C03563=1013.898,264.912,-139.732,168.814,53.259,160.172
C03564=1013.893,264.664,-139.704,168.809,53.267,160.173
C03565=1013.887,264.419,-139.676,168.803,53.274,160.173
C03566=1013.882,264.174,-139.648,168.798,53.282,160.174
C03567=1013.877,263.928,-139.620,168.793,53.290,160.175
C03568=1013.871,263.683,-139.592,168.787,53.298,160.175
C03569=1013.865,263.438,-139.565,168.782,53.306,160.176
C03570=1013.860,263.193,-139.538,168.777,53.313,160.177
C03571=1013.855,262.948,-139.510,168.772,53.321,160.177
C03572=1013.850,262.702,-139.482,168.766,53.329,160.178
C03573=1013.844,262.454,-139.454,168.762,53.337,160.179
C03574=1013.838,262.206,-139.426,168.756,53.346,160.179
C03575=1013.833,261.958,-139.398,168.751,53.353,160.180
C03576=1013.828,261.709,-139.371,168.746,53.361,160.181
C03577=1013.823,261.461,-139.343,168.740,53.369,160.181
C03578=1013.817,261.212,-139.315,168.735,53.377,160.182
C03579=1013.811,260.964,-139.287,168.729,53.386,160.183
C03580=1013.806,260.715,-139.259,168.725,53.393,160.183
C03581=1013.801,260.466,-139.231,168.719,53.402,160.184
C03582=1013.795,260.217,-139.203,168.714,53.410,160.185
C03583=1013.790,259.968,-139.175,168.708,53.418,160.185
C03584=1013.785,259.718,-139.147,168.703,53.426,160.186
C03585=1013.780,259.470,-139.119,168.699,53.434,160.187
C03586=1013.774,259.221,-139.092,168.693,53.443,160.188
C03587=1013.768,258.973,-139.064,168.687,53.451,160.188
C03588=1013.763,258.725,-139.037,168.682,53.459,160.189
C03589=1013.758,258.476,-139.011,168.677,53.468,160.190
C03590=1013.752,258.228,-138.983,168.672,53.476,160.191
C03591=1013.746,257.979,-138.956,168.666,53.484,160.191
C03592=1013.741,257.731,-138.928,168.662,53.492,160.192
C03593=1013.736,257.482,-138.900,168.656,53.501,160.193
C03594=1013.730,257.234,-138.874,168.651,53.509,160.194
C03595=1013.724,256.986,-138.846,168.646,53.518,160.194
C03596=1013.719,256.738,-138.819,168.640,53.526,160.195
C03597=1013.714,256.489,-138.792,168.635,53.534,160.196
C03598=1013.708,256.240,-138.764,168.630,53.543,160.197
C03599=1013.702,255.992,-138.737,168.625,53.551,160.197
C03600=1013.697,255.743,-138.710,168.620,53.560,160.198
C03601=1013.691,255.495,-138.683,168.614,53.568,160.199
C03602=1013.686,255.246,-138.656,168.610,53.576,160.200
C03603=1013.681,254.998,-138.629,168.604,53.585,160.200
C03604=1013.675,254.750,-138.601,168.599,53.593,160.201
C03605=1013.670,254.501,-138.574,168.594,53.602,160.202
C03606=1013.664,254.253,-138.547,168.589,53.610,160.203
C03607=1013.659,254.004,-138.520,168.583,53.619,160.204
C03608=1013.654,253.755,-138.493,168.578,53.628,160.204
C03609=1013.648,253.507,-138.466,168.573,53.635,160.205
C03610=1013.643,253.259,-138.438,168.568,53.644,160.206
C03611=1013.637,253.011,-138.412,168.562,53.653,160.207
C03612=1013.632,252.762,-138.384,168.558,53.661,160.208
C03613=1013.626,252.514,-138.358,168.552,53.670,160.208
C03614=1013.621,252.265,-138.330,168.548,53.678,160.209
C03615=1013.616,252.016,-138.303,168.542,53.687,160.210
C03616=1013.611,251.768,-138.276,168.537,53.696,160.211
C03617=1013.605,251.519,-138.249,168.532,53.704,160.212
C03618=1013.600,251.271,-138.223,168.527,53.713,160.212
C03619=1013.595,251.022,-138.195,168.522,53.721,160.213
C03620=1013.590,250.774,-138.168,168.517,53.730,160.214
C03621=1013.584,250.525,-138.141,168.511,53.739,160.215
C03622=1013.579,250.277,-138.114,168.507,53.747,160.216
C03623=1013.574,250.029,-138.088,168.501,53.756,160.216
C03624=1013.569,249.780,-138.061,168.496,53.765,160.217
C03625=1013.564,249.534,-138.034,168.491,53.773,160.218
C03626=1013.558,249.289,-138.007,168.486,53.782,160.219
C03627=1013.554,249.043,-137.981,168.482,53.791,160.220
C03628=1013.548,248.798,-137.954,168.476,53.799,160.220
C03629=1013.543,248.551,-137.928,168.472,53.808,160.221
C03630=1013.537,248.307,-137.901,168.466,53.817,160.222
C03631=1013.532,248.060,-137.875,168.460,53.825,160.223
C03632=1013.527,247.814,-137.849,168.456,53.834,160.224
C03633=1013.522,247.566,-137.821,168.451,53.843,160.225
C03634=1013.517,247.318,-137.794,168.447,53.851,160.226
C03635=1013.512,247.069,-137.768,168.441,53.860,160.226
C03636=1013.507,246.821,-137.741,168.435,53.869,160.227
C03637=1013.501,246.572,-137.715,168.431,53.877,160.228
C03638=1013.497,246.324,-137.688,168.426,53.886,160.229
C03639=1013.491,246.075,-137.661,168.421,53.895,160.230
C03640=1013.486,245.827,-137.634,168.416,53.904,160.231
C03641=1013.481,245.577,-137.607,168.411,53.913,160.231
C03642=1013.476,245.330,-137.581,168.406,53.922,160.232
C03643=1013.471,245.081,-137.554,168.400,53.931,160.233
C03644=1013.465,244.832,-137.528,168.396,53.940,160.234
C03645=1013.460,244.583,-137.501,168.390,53.948,160.235
C03646=1013.455,244.336,-137.474,168.385,53.957,160.236
C03647=1013.451,244.086,-137.448,168.381,53.966,160.237
C03648=1013.445,243.838,-137.421,168.375,53.975,160.237
C03649=1013.440,243.590,-137.394,168.370,53.984,160.238
C03650=1013.436,243.341,-137.368,168.366,53.993,160.239
C03651=1013.430,243.092,-137.341,168.361,54.002,160.240
C03652=1013.425,242.845,-137.314,168.355,54.011,160.241
C03653=1013.421,242.595,-137.288,168.350,54.020,160.242
C03654=1013.415,242.347,-137.261,168.346,54.029,160.243
C03655=1013.410,242.099,-137.236,168.341,54.038,160.244
C03656=1013.404,241.850,-137.209,168.336,54.047,160.245
C03657=1013.400,241.602,-137.183,168.330,54.057,160.245
C03658=1013.395,241.353,-137.157,168.325,54.066,160.246
C03659=1013.389,241.104,-137.130,168.321,54.075,160.248
C03660=1013.384,240.856,-137.105,168.316,54.084,160.248
C03661=1013.379,240.607,-137.077,168.311,54.093,160.249
C03662=1013.374,240.359,-137.052,168.306,54.102,160.250
C03663=1013.369,240.110,-137.026,168.300,54.111,160.251
C03664=1013.364,239.861,-136.999,168.296,54.121,160.252
C03665=1013.359,239.613,-136.973,168.291,54.130,160.253
C03666=1013.353,239.364,-136.947,168.286,54.139,160.254
C03667=1013.348,239.116,-136.922,168.281,54.149,160.255
C03668=1013.343,238.867,-136.894,168.276,54.158,160.256
C03669=1013.338,238.618,-136.868,168.271,54.167,160.257
C03670=1013.333,238.370,-136.843,168.266,54.177,160.258
C03671=1013.328,238.121,-136.817,168.262,54.185,160.259
C03672=1013.323,237.873,-136.791,168.257,54.194,160.259
C03673=1013.317,237.624,-136.765,168.252,54.204,160.261
C03674=1013.312,237.376,-136.739,168.247,54.213,160.261
C03675=1013.307,237.127,-136.713,168.242,54.223,160.262
C03676=1013.302,236.879,-136.688,168.237,54.232,160.263
C03677=1013.296,236.630,-136.662,168.232,54.242,160.264
C03678=1013.291,236.382,-136.636,168.227,54.251,160.265
C03679=1013.286,236.133,-136.610,168.222,54.261,160.266
C03680=1013.281,235.884,-136.585,168.217,54.270,160.267
C03681=1013.276,235.635,-136.559,168.212,54.280,160.268
C03682=1013.271,235.387,-136.533,168.207,54.289,160.269
C03683=1013.265,235.138,-136.507,168.202,54.299,160.270
C03684=1013.260,234.890,-136.482,168.197,54.309,160.271
C03685=1013.256,234.641,-136.457,168.192,54.318,160.272
C03686=1013.250,234.392,-136.431,168.187,54.328,160.273
C03687=1013.245,234.144,-136.405,168.182,54.337,160.274
C03688=1013.240,233.895,-136.379,168.177,54.347,160.275
C03689=1013.235,233.644,-136.353,168.172,54.356,160.276
C03690=1013.230,233.394,-136.328,168.168,54.366,160.277
C03691=1013.225,233.143,-136.302,168.163,54.375,160.278
C03692=1013.220,232.892,-136.276,168.158,54.385,160.279
C03693=1013.214,232.644,-136.251,168.153,54.395,160.280
C03694=1013.209,232.396,-136.225,168.148,54.405,160.281
C03695=1013.204,232.147,-136.200,168.143,54.414,160.282
C03696=1013.199,231.898,-136.175,168.138,54.424,160.283
C03697=1013.194,231.649,-136.149,168.134,54.434,160.284
C03698=1013.189,231.401,-136.123,168.129,54.443,160.285
C03699=1013.184,231.152,-136.098,168.124,54.453,160.286
C03700=1013.179,230.903,-136.073,168.119,54.463,160.287
C03701=1013.174,230.655,-136.047,168.114,54.472,160.288
C03702=1013.169,230.406,-136.021,168.110,54.482,160.290
C03703=1013.164,230.158,-135.996,168.104,54.491,160.290
C03704=1013.159,229.909,-135.971,168.100,54.501,160.291
C03705=1013.154,229.660,-135.945,168.095,54.511,160.293
C03706=1013.149,229.412,-135.919,168.090,54.521,160.294
C03707=1013.144,229.163,-135.895,168.086,54.531,160.295
C03708=1013.139,228.915,-135.869,168.080,54.541,160.296
C03709=1013.134,228.665,-135.844,168.075,54.550,160.296
C03710=1013.129,228.417,-135.819,168.070,54.560,160.298
C03711=1013.124,228.168,-135.794,168.065,54.570,160.299
C03712=1013.118,227.919,-135.768,168.061,54.580,160.300
C03713=1013.114,227.670,-135.744,168.056,54.590,160.301
C03714=1013.109,227.422,-135.718,168.051,54.600,160.302
C03715=1013.104,227.173,-135.693,168.047,54.610,160.303
C03716=1013.099,226.925,-135.668,168.042,54.619,160.304
C03717=1013.093,226.676,-135.643,168.036,54.630,160.305
C03718=1013.089,226.427,-135.617,168.032,54.640,160.306
C03719=1013.084,226.178,-135.593,168.027,54.649,160.307
C03720=1013.079,225.930,-135.567,168.022,54.659,160.308
C03721=1013.074,225.682,-135.543,168.018,54.669,160.309
C03722=1013.069,225.432,-135.518,168.013,54.679,160.311
C03723=1013.063,225.184,-135.493,168.008,54.690,160.312
C03724=1013.058,224.935,-135.468,168.003,54.700,160.313
C03725=1013.053,224.686,-135.443,167.999,54.710,160.314
C03726=1013.049,224.438,-135.419,167.994,54.720,160.315
C03727=1013.043,224.190,-135.394,167.989,54.730,160.316
C03728=1013.038,223.941,-135.369,167.984,54.740,160.317
C03729=1013.033,223.691,-135.344,167.979,54.751,160.318
C03730=1013.028,223.443,-135.319,167.975,54.761,160.319
C03731=1013.023,223.194,-135.295,167.970,54.770,160.321
C03732=1013.018,222.946,-135.269,167.964,54.781,160.321
C03733=1013.013,222.697,-135.245,167.960,54.791,160.323
C03734=1013.008,222.448,-135.220,167.956,54.801,160.324
C03735=1013.003,222.200,-135.196,167.951,54.811,160.325
C03736=1012.998,221.951,-135.171,167.945,54.822,160.326
C03737=1012.993,221.702,-135.147,167.941,54.832,160.327
C03738=1012.988,221.452,-135.122,167.937,54.842,160.328
C03739=1012.982,221.204,-135.098,167.931,54.852,160.329
C03740=1012.978,220.956,-135.072,167.927,54.863,160.331
C03741=1012.972,220.707,-135.048,167.922,54.873,160.332
C03742=1012.968,220.458,-135.023,167.918,54.883,160.333
C03743=1012.962,220.210,-134.999,167.912,54.894,160.334
C03744=1012.958,219.961,-134.974,167.908,54.904,160.335
C03745=1012.952,219.712,-134.950,167.903,54.914,160.336
C03746=1012.948,219.463,-134.925,167.898,54.925,160.337
C03747=1012.943,219.215,-134.900,167.894,54.935,160.339
C03748=1012.938,218.966,-134.876,167.889,54.945,160.340
C03749=1012.933,218.706,-134.850,167.884,54.956,160.341
C03750=1012.927,218.447,-134.825,167.879,54.967,160.342
C03751=1012.923,218.189,-134.799,167.875,54.978,160.343
C03752=1012.918,217.929,-134.774,167.869,54.989,160.345
C03753=1012.913,217.681,-134.749,167.865,54.999,160.346
C03754=1012.908,217.432,-134.724,167.860,55.010,160.347
C03755=1012.903,217.183,-134.701,167.855,55.020,160.348
C03756=1012.898,216.934,-134.677,167.851,55.030,160.349
C03757=1012.892,216.686,-134.652,167.846,55.041,160.350
C03758=1012.888,216.437,-134.627,167.841,55.051,160.352
C03759=1012.883,216.188,-134.604,167.836,55.062,160.353
C03760=1012.878,215.939,-134.580,167.832,55.072,160.354
C03761=1012.872,215.690,-134.555,167.827,55.083,160.355
C03762=1012.867,215.442,-134.531,167.822,55.093,160.356
C03763=1012.863,215.193,-134.507,167.818,55.104,160.358
C03764=1012.858,214.944,-134.483,167.813,55.115,160.359
C03765=1012.853,214.696,-134.459,167.808,55.125,160.360
C03766=1012.848,214.447,-134.435,167.803,55.136,160.361
C03767=1012.842,214.198,-134.411,167.799,55.147,160.362
C03768=1012.838,213.948,-134.387,167.794,55.157,160.363
C03769=1012.833,213.700,-134.363,167.790,55.168,160.365
C03770=1012.828,213.451,-134.338,167.785,55.179,160.366
C03771=1012.823,213.203,-134.315,167.780,55.189,160.367
C03772=1012.819,212.954,-134.290,167.775,55.200,160.368
C03773=1012.814,212.705,-134.267,167.771,55.211,160.370
C03774=1012.808,212.456,-134.243,167.765,55.221,160.371
C03775=1012.803,212.207,-134.218,167.761,55.232,160.372
C03776=1012.798,211.958,-134.195,167.757,55.243,160.373
C03777=1012.794,211.710,-134.170,167.752,55.254,160.375
C03778=1012.789,211.461,-134.147,167.748,55.264,160.376
C03779=1012.784,211.212,-134.123,167.743,55.275,160.377
C03780=1012.779,210.963,-134.099,167.739,55.286,160.378
C03781=1012.774,210.714,-134.075,167.734,55.297,160.379
C03782=1012.770,210.466,-134.051,167.730,55.308,160.381
C03783=1012.765,210.217,-134.027,167.724,55.318,160.382
C03784=1012.760,209.968,-134.003,167.719,55.329,160.383
C03785=1012.755,209.719,-133.980,167.715,55.340,160.384
C03786=1012.750,209.471,-133.956,167.710,55.351,160.385
C03787=1012.746,209.221,-133.932,167.706,55.362,160.387
C03788=1012.740,208.973,-133.907,167.701,55.373,160.388
C03789=1012.736,208.724,-133.884,167.697,55.384,160.389
C03790=1012.731,208.475,-133.861,167.692,55.395,160.391
C03791=1012.726,208.226,-133.836,167.688,55.405,160.392
C03792=1012.721,207.977,-133.813,167.682,55.416,160.393
C03793=1012.716,207.729,-133.790,167.677,55.427,160.394
C03794=1012.711,207.479,-133.766,167.673,55.438,160.395
C03795=1012.706,207.231,-133.742,167.668,55.449,160.397
C03796=1012.702,206.982,-133.719,167.664,55.460,160.398
C03797=1012.697,206.733,-133.695,167.659,55.471,160.399
C03798=1012.692,206.484,-133.672,167.654,55.482,160.400
C03799=1012.687,206.235,-133.648,167.650,55.493,160.402
C03800=1012.682,205.987,-133.624,167.646,55.505,160.403
C03801=1012.676,205.738,-133.601,167.641,55.516,160.405
C03802=1012.672,205.489,-133.578,167.637,55.527,160.406
C03803=1012.667,205.240,-133.555,167.632,55.538,160.407
C03804=1012.662,204.992,-133.531,167.627,55.549,160.408
C03805=1012.657,204.743,-133.508,167.623,55.560,160.410
C03806=1012.652,204.493,-133.484,167.618,55.571,160.411
C03807=1012.648,204.245,-133.461,167.613,55.582,160.412
C03808=1012.643,203.996,-133.438,167.609,55.593,160.413
C03809=1012.637,203.731,-133.413,167.604,55.605,160.415
C03810=1012.632,203.465,-133.388,167.599,55.617,160.416
C03811=1012.627,203.201,-133.364,167.595,55.629,160.418
C03812=1012.622,202.936,-133.339,167.590,55.641,160.419
C03813=1012.604,201.768,-133.238,167.040,55.554,160.267
C03814=1012.600,201.520,-133.216,167.036,55.567,160.269
C03815=1012.597,201.270,-133.194,167.030,55.579,160.270
C03816=1012.593,201.021,-133.174,167.026,55.592,160.272
C03817=1012.589,200.773,-133.151,167.022,55.604,160.273
C03818=1012.585,200.523,-133.130,167.016,55.616,160.274
C03819=1012.582,200.274,-133.109,167.012,55.629,160.276
C03820=1012.578,200.025,-133.087,167.008,55.641,160.277
C03821=1012.575,199.776,-133.066,167.003,55.654,160.279
C03822=1012.570,199.527,-133.044,166.998,55.666,160.280
C03823=1012.567,199.278,-133.023,166.994,55.678,160.282
C03824=1012.563,199.029,-133.001,166.989,55.690,160.283
C03825=1012.560,198.780,-132.980,166.984,55.703,160.285
C03826=1012.556,198.530,-132.959,166.980,55.715,160.286
C03827=1012.552,198.281,-132.938,166.975,55.727,160.288
C03828=1012.548,198.033,-132.917,166.970,55.740,160.289
C03829=1012.543,197.783,-132.896,166.966,55.752,160.290
C03830=1012.540,197.534,-132.875,166.962,55.765,160.292
C03831=1012.536,197.285,-132.854,166.956,55.778,160.293
C03832=1012.532,197.036,-132.833,166.952,55.790,160.295
C03833=1012.529,196.787,-132.811,166.948,55.802,160.296
C03834=1012.525,196.538,-132.790,166.943,55.815,160.298
C03835=1012.521,196.290,-132.770,166.938,55.827,160.299
C03836=1012.517,196.039,-132.749,166.934,55.840,160.301
C03837=1012.513,195.790,-132.728,166.930,55.852,160.302
C03838=1012.509,195.542,-132.707,166.925,55.865,160.304
C03839=1012.506,195.293,-132.686,166.920,55.877,160.305
C03840=1012.502,195.043,-132.665,166.917,55.890,160.307
C03841=1012.498,194.794,-132.644,166.912,55.902,160.308
C03842=1012.494,194.546,-132.623,166.907,55.914,160.309
C03843=1012.490,194.296,-132.603,166.903,55.927,160.311
C03844=1012.487,194.047,-132.581,166.898,55.939,160.312
C03845=1012.483,193.798,-132.560,166.894,55.952,160.314
C03846=1012.599,214.705,-134.836,167.768,55.269,160.382
C03847=1012.605,215.007,-134.865,167.774,55.256,160.380
C03848=1012.611,215.309,-134.895,167.779,55.243,160.379
C03849=1012.617,215.611,-134.924,167.786,55.230,160.377
C03850=1012.623,215.913,-134.953,167.791,55.218,160.376
C03851=1012.628,216.162,-134.977,167.796,55.207,160.375
C03852=1012.633,216.411,-135.001,167.800,55.196,160.374
C03853=1012.638,216.660,-135.026,167.805,55.186,160.372
C03854=1012.643,216.908,-135.050,167.810,55.175,160.371
C03855=1012.648,217.157,-135.073,167.815,55.165,160.370
C03856=1012.653,217.405,-135.097,167.820,55.154,160.369
C03857=1012.658,217.654,-135.122,167.824,55.144,160.368
C03858=1012.663,217.903,-135.146,167.828,55.134,160.366
C03859=1012.668,218.165,-135.172,167.833,55.123,160.365
C03860=1012.673,218.426,-135.198,167.838,55.111,160.364
C03861=1012.678,218.688,-135.223,167.844,55.101,160.363
C03862=1012.682,218.949,-135.249,167.849,55.090,160.362
C03863=1012.688,219.198,-135.273,167.853,55.079,160.360
C03864=1012.692,219.447,-135.298,167.858,55.069,160.359
C03865=1012.698,219.695,-135.323,167.863,55.059,160.358
C03866=1012.702,219.944,-135.347,167.867,55.048,160.357
C03867=1012.707,220.193,-135.372,167.872,55.038,160.356
C03868=1012.712,220.442,-135.396,167.878,55.028,160.355
C03869=1012.717,220.690,-135.421,167.882,55.017,160.354
C03870=1012.722,220.939,-135.446,167.886,55.007,160.353
C03871=1012.727,221.188,-135.470,167.892,54.997,160.352
C03872=1012.732,221.437,-135.495,167.896,54.987,160.351
C03873=1012.737,221.685,-135.519,167.901,54.976,160.349
C03874=1012.742,221.934,-135.544,167.906,54.966,160.348
C03875=1012.747,222.183,-135.568,167.911,54.956,160.347
C03876=1012.751,222.431,-135.593,167.915,54.946,160.346
C03877=1012.757,222.680,-135.617,167.919,54.935,160.345
C03878=1012.761,222.929,-135.642,167.925,54.925,160.344
C03879=1012.767,223.178,-135.666,167.930,54.915,160.343
C03880=1012.771,223.426,-135.692,167.934,54.905,160.342
C03881=1012.777,223.675,-135.716,167.940,54.895,160.341
C03882=1012.782,223.924,-135.741,167.944,54.884,160.339
C03883=1012.787,224.173,-135.766,167.949,54.874,160.338
C03884=1012.792,224.422,-135.790,167.953,54.864,160.337
C03885=1012.797,224.670,-135.815,167.959,54.854,160.336
C03886=1012.802,224.919,-135.840,167.964,54.844,160.335
C03887=1012.807,225.167,-135.864,167.968,54.834,160.334
C03888=1012.812,225.416,-135.889,167.973,54.824,160.333
C03889=1012.817,225.664,-135.914,167.978,54.814,160.332
C03890=1012.822,225.913,-135.939,167.983,54.803,160.331
C03891=1012.827,226.162,-135.964,167.987,54.793,160.329
C03892=1012.832,226.411,-135.989,167.992,54.784,160.328
C03893=1012.837,226.659,-136.014,167.996,54.774,160.327
C03894=1012.842,226.908,-136.039,168.002,54.763,160.326
C03895=1012.846,227.157,-136.064,168.007,54.753,160.325
C03896=1012.851,227.405,-136.089,168.012,54.744,160.324
C03897=1012.857,227.654,-136.114,168.017,54.734,160.323
C03898=1012.862,227.903,-136.140,168.021,54.724,160.322
C03899=1012.867,228.152,-136.165,168.026,54.714,160.321
C03900=1012.871,228.400,-136.190,168.032,54.704,160.320
C03901=1012.877,228.649,-136.214,168.036,54.694,160.319
C03902=1012.882,228.898,-136.240,168.041,54.684,160.318
C03903=1012.887,229.146,-136.265,168.045,54.674,160.317
C03904=1012.892,229.395,-136.291,168.050,54.665,160.316
C03905=1012.896,229.644,-136.316,168.055,54.655,160.315
C03906=1012.901,229.892,-136.341,168.060,54.646,160.314
C03907=1012.906,230.142,-136.366,168.065,54.636,160.313
C03908=1012.911,230.390,-136.392,168.070,54.625,160.312
C03909=1012.917,230.638,-136.417,168.075,54.615,160.311
C03910=1012.921,230.887,-136.442,168.080,54.606,160.310
C03911=1012.927,231.136,-136.468,168.085,54.596,160.309
C03912=1012.932,231.384,-136.493,168.090,54.587,160.308
C03913=1012.936,231.633,-136.518,168.094,54.577,160.307
C03914=1012.942,231.882,-136.544,168.099,54.567,160.306
C03915=1012.946,232.130,-136.570,168.104,54.558,160.305
C03916=1012.951,232.379,-136.594,168.109,54.548,160.304
C03917=1012.957,232.628,-136.620,168.113,54.538,160.303
C03918=1012.961,232.876,-136.646,168.119,54.529,160.302
C03919=1012.967,233.130,-136.671,168.123,54.519,160.301
C03920=1012.972,233.382,-136.698,168.129,54.509,160.300
C03921=1012.977,233.635,-136.723,168.134,54.499,160.299
C03922=1012.982,233.887,-136.750,168.138,54.489,160.298
C03923=1012.987,234.136,-136.775,168.144,54.480,160.297
C03924=1012.992,234.385,-136.801,168.148,54.470,160.296
C03925=1012.997,234.633,-136.825,168.154,54.461,160.295
C03926=1013.003,234.882,-136.851,168.158,54.451,160.294
C03927=1013.008,235.131,-136.877,168.163,54.441,160.293
C03928=1013.013,235.379,-136.903,168.168,54.432,160.292
C03929=1013.018,235.628,-136.928,168.173,54.422,160.291
C03930=1013.023,235.876,-136.954,168.178,54.413,160.290
C03931=1013.028,236.125,-136.980,168.183,54.403,160.289
C03932=1013.033,236.374,-137.005,168.188,54.394,160.288
C03933=1013.038,236.623,-137.031,168.193,54.384,160.287
C03934=1013.043,236.871,-137.056,168.198,54.375,160.286
C03935=1013.049,237.120,-137.082,168.203,54.365,160.285
C03936=1013.054,237.369,-137.108,168.208,54.356,160.284
C03937=1013.059,237.618,-137.134,168.213,54.346,160.283
C03938=1013.064,237.866,-137.159,168.218,54.337,160.282
C03939=1013.069,238.114,-137.185,168.223,54.327,160.281
C03940=1013.075,238.362,-137.212,168.228,54.318,160.280
C03941=1013.079,238.611,-137.238,168.232,54.308,160.279
C03942=1013.084,238.860,-137.264,168.238,54.299,160.278
C03943=1013.089,239.108,-137.289,168.243,54.290,160.277
C03944=1013.095,239.357,-137.315,168.248,54.281,160.277
C03945=1013.099,239.605,-137.342,168.253,54.271,160.275
C03946=1013.104,239.854,-137.368,168.257,54.262,160.274
C03947=1013.110,240.103,-137.394,168.262,54.253,160.274
C03948=1013.114,240.352,-137.420,168.267,54.243,160.273
C03949=1013.120,240.600,-137.447,168.272,54.234,160.272
C03950=1013.125,240.848,-137.472,168.278,54.225,160.271
C03951=1013.130,241.097,-137.498,168.283,54.216,160.270
C03952=1013.134,241.346,-137.524,168.288,54.206,160.269
C03953=1013.140,241.594,-137.551,168.293,54.197,160.268
C03954=1013.145,241.843,-137.577,168.298,54.188,160.267
C03955=1013.150,242.092,-137.603,168.302,54.179,160.266
C03956=1013.155,242.340,-137.630,168.308,54.170,160.265
C03957=1013.160,242.589,-137.655,168.313,54.161,160.265
C03958=1013.165,242.837,-137.683,168.318,54.151,160.263
C03959=1013.170,243.085,-137.708,168.323,54.142,160.263
C03960=1013.175,243.334,-137.735,168.327,54.134,160.262
C03961=1013.181,243.583,-137.762,168.332,54.125,160.261
C03962=1013.185,243.831,-137.788,168.338,54.115,160.260
C03963=1013.190,244.080,-137.815,168.343,54.106,160.259
C03964=1013.196,244.329,-137.841,168.347,54.098,160.258
C03965=1013.200,244.577,-137.868,168.352,54.089,160.257
C03966=1013.206,244.826,-137.894,168.358,54.080,160.256
C03967=1013.211,245.074,-137.921,168.363,54.070,160.256
C03968=1013.215,245.322,-137.948,168.367,54.062,160.255
C03969=1013.220,245.571,-137.974,168.373,54.053,160.254
C03970=1013.225,245.820,-138.001,168.378,54.044,160.253
C03971=1013.231,246.068,-138.028,168.383,54.035,160.252
C03972=1013.235,246.317,-138.054,168.388,54.027,160.251
C03973=1013.241,246.565,-138.081,168.393,54.018,160.251
C03974=1013.246,246.813,-138.108,168.398,54.008,160.250
C03975=1013.251,247.062,-138.135,168.403,53.999,160.249
C03976=1013.256,247.311,-138.161,168.408,53.991,160.248
C03977=1013.261,247.560,-138.188,168.413,53.982,160.247
C03978=1013.266,247.807,-138.214,168.419,53.973,160.246
C03979=1013.271,248.055,-138.241,168.424,53.964,160.246
C03980=1013.276,248.302,-138.268,168.428,53.956,160.245
C03981=1013.281,248.550,-138.295,168.434,53.947,160.244
C03982=1013.287,248.797,-138.322,168.439,53.937,160.243
C03983=1013.292,249.045,-138.348,168.444,53.930,160.242
C03984=1013.297,249.291,-138.375,168.449,53.920,160.241
C03985=1013.302,249.538,-138.401,168.454,53.911,160.241
C03986=1013.308,249.786,-138.428,168.459,53.903,160.240
C03987=1013.313,250.034,-138.455,168.464,53.894,160.239
C03988=1013.318,250.283,-138.482,168.470,53.885,160.238
C03989=1013.323,250.531,-138.509,168.474,53.877,160.237
C03990=1013.328,250.781,-138.535,168.480,53.868,160.237
C03991=1013.333,251.028,-138.562,168.485,53.859,160.236
C03992=1013.338,251.277,-138.589,168.489,53.851,160.235
C03993=1013.344,251.525,-138.616,168.495,53.842,160.234
C03994=1013.349,251.774,-138.643,168.500,53.833,160.233
C03995=1013.354,252.023,-138.670,168.506,53.824,160.232
C03996=1013.360,252.271,-138.697,168.510,53.816,160.232
C03997=1013.365,252.520,-138.724,168.516,53.807,160.231
C03998=1013.371,252.768,-138.751,168.521,53.798,160.230
C03999=1013.376,253.017,-138.778,168.526,53.790,160.229
C04000=1013.381,253.265,-138.805,168.531,53.781,160.228
C04001=1013.387,253.514,-138.832,168.537,53.773,160.228
C04002=1013.392,253.762,-138.859,168.541,53.764,160.227
C04003=1013.397,254.011,-138.886,168.547,53.756,160.226
C04004=1013.403,254.259,-138.914,168.552,53.747,160.225
C04005=1013.408,254.507,-138.941,168.557,53.738,160.224
C04006=1013.414,254.756,-138.968,168.562,53.730,160.224
C04007=1013.419,255.004,-138.995,168.568,53.721,160.223
C04008=1013.424,255.253,-139.021,168.573,53.713,160.222
C04009=1013.429,255.501,-139.049,168.578,53.704,160.221
C04010=1013.434,255.750,-139.076,168.584,53.696,160.221
C04011=1013.441,255.998,-139.103,168.588,53.687,160.220
C04012=1013.446,256.247,-139.131,168.594,53.679,160.219
C04013=1013.451,256.495,-139.157,168.600,53.671,160.219
C04014=1013.456,256.744,-139.184,168.604,53.662,160.218
C04015=1013.461,256.992,-139.212,168.610,53.654,160.217
C04016=1013.468,257.240,-139.239,168.614,53.645,160.216
C04017=1013.473,257.489,-139.266,168.620,53.637,160.215
C04018=1013.478,257.737,-139.293,168.625,53.628,160.215
C04019=1013.484,257.986,-139.321,168.630,53.620,160.214
C04020=1013.490,258.234,-139.348,168.636,53.612,160.213
C04021=1013.495,258.483,-139.375,168.641,53.603,160.212
C04022=1013.500,258.731,-139.402,168.646,53.595,160.212
C04023=1013.506,258.979,-139.430,168.652,53.586,160.211
C04024=1013.511,259.228,-139.457,168.657,53.577,160.210
C04025=1013.517,259.476,-139.485,168.662,53.570,160.209
C04026=1013.522,259.725,-139.512,168.668,53.561,160.209
C04027=1013.527,259.973,-139.540,168.673,53.553,160.208
C04028=1013.532,260.221,-139.568,168.678,53.545,160.207
C04029=1013.538,260.470,-139.596,168.683,53.537,160.207
C04030=1013.543,260.718,-139.624,168.689,53.529,160.206
C04031=1013.548,260.967,-139.651,168.694,53.521,160.205
C04032=1013.554,261.215,-139.679,168.699,53.512,160.205
C04033=1013.559,261.463,-139.707,168.704,53.504,160.204
C04034=1013.565,261.712,-139.734,168.710,53.496,160.203
C04035=1013.570,261.960,-139.762,168.715,53.488,160.202
C04036=1013.575,262.208,-139.790,168.720,53.480,160.202
C04037=1013.581,262.456,-139.818,168.725,53.472,160.201
C04038=1013.586,262.705,-139.846,168.731,53.464,160.200
C04039=1013.592,262.951,-139.873,168.736,53.456,160.200
C04040=1013.597,263.198,-139.901,168.741,53.448,160.199
C04041=1013.602,263.444,-139.929,168.747,53.440,160.198
C04042=1013.608,263.690,-139.957,168.752,53.432,160.198
C04043=1013.613,263.937,-139.984,168.758,53.424,160.197
C04044=1013.619,264.182,-140.012,168.763,53.416,160.197
C04045=1013.624,264.429,-140.040,168.768,53.408,160.196
C04046=1013.629,264.675,-140.068,168.773,53.400,160.195
C04047=1013.635,264.923,-140.096,168.778,53.392,160.194
C04048=1013.640,265.171,-140.124,168.784,53.384,160.194
C04049=1013.645,265.421,-140.153,168.789,53.377,160.193
C04050=1013.651,265.669,-140.181,168.795,53.368,160.193
C04051=1013.656,265.917,-140.208,168.800,53.361,160.192
C04052=1013.662,266.165,-140.237,168.806,53.352,160.191
C04053=1013.667,266.413,-140.265,168.811,53.345,160.191
C04054=1013.673,266.661,-140.293,168.816,53.337,160.190
C04055=1013.678,266.911,-140.322,168.822,53.329,160.190
C04056=1013.683,267.159,-140.350,168.827,53.321,160.189
C04057=1013.688,267.407,-140.378,168.833,53.314,160.188
C04058=1013.694,267.655,-140.406,168.838,53.306,160.188
C04059=1013.700,267.903,-140.434,168.843,53.298,160.187
C04060=1013.705,268.153,-140.463,168.848,53.290,160.186
C04061=1013.710,268.401,-140.491,168.854,53.283,160.186
C04062=1013.716,268.648,-140.519,168.860,53.274,160.185
C04063=1013.722,268.897,-140.548,168.865,53.267,160.185
C04064=1013.726,269.145,-140.576,168.870,53.259,160.184
C04065=1013.732,269.394,-140.605,168.876,53.251,160.183
C04066=1013.738,269.641,-140.633,168.881,53.244,160.183
C04067=1013.743,269.890,-140.662,168.886,53.236,160.182
C04068=1013.749,270.138,-140.690,168.892,53.229,160.182
C04069=1013.753,270.387,-140.719,168.897,53.221,160.181
C04070=1013.759,270.635,-140.748,168.903,53.213,160.181
C04071=1013.765,270.883,-140.776,168.908,53.205,160.180
C04072=1013.770,271.132,-140.805,168.914,53.198,160.179
C04073=1013.776,271.379,-140.833,168.919,53.190,160.179
C04074=1013.782,271.628,-140.862,168.925,53.183,160.178
C04075=1013.787,271.876,-140.891,168.930,53.175,160.177
C04076=1013.792,272.125,-140.919,168.936,53.167,160.177
C04077=1013.797,272.372,-140.948,168.941,53.160,160.177
C04078=1013.803,272.621,-140.977,168.946,53.152,160.176
C04079=1013.809,272.870,-141.006,168.953,53.145,160.175
C04080=1013.814,273.118,-141.034,168.958,53.138,160.175
C04081=1013.820,273.366,-141.063,168.963,53.130,160.174
C04082=1013.825,273.614,-141.092,168.969,53.122,160.174
C04083=1013.831,273.862,-141.121,168.974,53.115,160.173
C04084=1013.836,274.111,-141.150,168.979,53.108,160.172
C04085=1013.842,274.359,-141.179,168.986,53.100,160.172
C04086=1013.847,274.608,-141.208,168.991,53.093,160.172
C04087=1013.853,274.855,-141.236,168.996,53.086,160.171
C04088=1013.858,275.104,-141.266,169.002,53.078,160.170
C04089=1013.864,275.352,-141.294,169.007,53.070,160.170
C04090=1013.869,275.600,-141.323,169.013,53.063,160.169
C04091=1013.876,275.848,-141.352,169.018,53.056,160.169
C04092=1013.881,276.096,-141.382,169.025,53.049,160.169
C04093=1013.886,276.345,-141.410,169.029,53.041,160.168
C04094=1013.892,276.593,-141.440,169.035,53.034,160.167
C04095=1013.897,276.841,-141.469,169.040,53.027,160.167
C04096=1013.902,277.089,-141.499,169.046,53.019,160.166
C04097=1013.909,277.338,-141.528,169.052,53.012,160.166
C04098=1013.914,277.586,-141.557,169.057,53.005,160.165
C04099=1013.920,277.889,-141.592,169.064,52.996,160.165
C04100=1013.927,278.192,-141.629,169.071,52.988,160.164
C04101=1013.934,278.495,-141.664,169.077,52.978,160.164
C04102=1013.941,278.798,-141.700,169.084,52.970,160.163
C04103=1013.946,279.046,-141.730,169.091,52.962,160.163
C04104=1013.953,279.295,-141.759,169.096,52.955,160.162
C04105=1013.958,279.543,-141.789,169.101,52.948,160.162
C04106=1013.963,279.791,-141.818,169.107,52.941,160.161
C04107=1013.968,280.039,-141.847,169.113,52.934,160.161
C04108=1013.975,280.287,-141.877,169.118,52.927,160.160
C04109=1013.980,280.536,-141.906,169.124,52.920,160.160
C04110=1013.986,280.784,-141.936,169.130,52.913,160.159
C04111=1013.991,281.032,-141.964,169.136,52.906,160.159
C04112=1013.997,281.280,-141.994,169.141,52.898,160.158
C04113=1014.002,281.529,-142.024,169.147,52.891,160.158
C04114=1014.008,281.777,-142.053,169.152,52.884,160.157
C04115=1014.014,282.025,-142.082,169.158,52.878,160.157
C04116=1014.020,282.273,-142.113,169.164,52.870,160.157
C04117=1014.026,282.521,-142.142,169.170,52.863,160.156
C04118=1014.031,282.769,-142.171,169.175,52.856,160.156
C04119=1014.037,283.017,-142.201,169.180,52.849,160.155
C04120=1014.042,283.266,-142.230,169.187,52.842,160.155
C04121=1014.048,283.513,-142.261,169.192,52.835,160.154
C04122=1014.054,283.762,-142.290,169.198,52.828,160.154
C04123=1014.060,284.010,-142.319,169.204,52.822,160.154
C04124=1014.065,284.259,-142.349,169.209,52.815,160.153
C04125=1014.071,284.506,-142.379,169.215,52.807,160.153
C04126=1014.077,284.755,-142.409,169.221,52.801,160.152
C04127=1014.082,285.003,-142.439,169.227,52.794,160.152
C04128=1014.088,285.251,-142.469,169.232,52.787,160.152
C04129=1014.094,285.499,-142.499,169.238,52.780,160.151
C04130=1014.099,285.747,-142.529,169.244,52.774,160.151
C04131=1014.105,285.968,-142.555,169.249,52.767,160.151
C04132=1014.110,286.189,-142.582,169.254,52.761,160.150
C04133=1014.115,286.410,-142.608,169.259,52.755,160.150
C04134=1014.120,286.631,-142.635,169.265,52.749,160.149
C04135=1014.125,286.852,-142.662,169.270,52.743,160.149
C04136=1014.130,287.073,-142.689,169.274,52.737,160.149
C04137=1014.135,287.293,-142.716,169.280,52.731,160.149
C04138=1014.140,287.514,-142.743,169.286,52.725,160.148
C04139=1014.145,287.762,-142.772,169.291,52.718,160.148
C04140=1014.151,288.010,-142.803,169.297,52.712,160.147
C04141=1014.157,288.258,-142.833,169.303,52.705,160.147
C04142=1014.163,288.507,-142.863,169.308,52.698,160.147
C04143=1014.169,288.755,-142.893,169.314,52.692,160.146
C04144=1014.175,289.003,-142.924,169.320,52.685,160.146
C04145=1014.181,289.251,-142.954,169.326,52.678,160.146
C04146=1014.186,289.499,-142.984,169.332,52.672,160.145
C04147=1014.192,289.747,-143.014,169.338,52.665,160.145
C04148=1014.198,289.995,-143.045,169.343,52.659,160.145
C04149=1014.203,290.242,-143.075,169.349,52.652,160.144
C04150=1014.210,290.492,-143.105,169.355,52.645,160.144
C04151=1014.215,290.739,-143.135,169.360,52.639,160.144
C04152=1014.221,290.987,-143.166,169.367,52.632,160.143
C04153=1014.226,291.235,-143.197,169.373,52.626,160.143
C04154=1014.232,291.483,-143.227,169.379,52.619,160.143
C04155=1014.238,291.731,-143.257,169.384,52.612,160.142
C04156=1014.244,291.979,-143.288,169.390,52.606,160.142
C04157=1014.250,292.227,-143.318,169.396,52.600,160.142
C04158=1014.256,292.475,-143.349,169.402,52.593,160.141
C04159=1014.261,292.736,-143.381,169.409,52.587,160.141
C04160=1014.268,292.998,-143.414,169.415,52.580,160.141
C04161=1014.273,293.259,-143.446,169.421,52.573,160.141
C04162=1014.280,293.520,-143.479,169.427,52.566,160.140
C04163=1014.285,293.768,-143.510,169.433,52.560,160.140
C04164=1014.291,294.016,-143.541,169.438,52.554,160.140
C04165=1014.296,294.264,-143.571,169.445,52.548,160.140
C04166=1014.303,294.512,-143.603,169.451,52.542,160.139
C04167=1014.308,294.760,-143.634,169.456,52.535,160.139
C04168=1014.313,295.008,-143.664,169.462,52.529,160.139
C04169=1014.319,295.256,-143.696,169.468,52.522,160.138
C04170=1014.325,295.504,-143.727,169.474,52.516,160.138
C04171=1014.330,295.752,-143.758,169.480,52.510,160.138
C04172=1014.336,295.999,-143.789,169.486,52.504,160.138
C04173=1014.342,296.248,-143.820,169.492,52.498,160.137
C04174=1014.348,296.496,-143.851,169.498,52.491,160.137
C04175=1014.353,296.744,-143.882,169.504,52.486,160.137
C04176=1014.360,296.992,-143.913,169.510,52.479,160.137
C04177=1014.365,297.240,-143.944,169.517,52.473,160.137
C04178=1014.371,297.487,-143.975,169.523,52.467,160.136
C04179=1014.377,297.736,-144.007,169.529,52.461,160.136
C04180=1014.383,297.983,-144.038,169.535,52.454,160.136
C04181=1014.389,298.232,-144.069,169.541,52.449,160.136
C04182=1014.395,298.479,-144.100,169.547,52.442,160.135
C04183=1014.400,298.727,-144.131,169.553,52.436,160.135
C04184=1014.406,298.975,-144.163,169.559,52.430,160.135
C04185=1014.412,299.223,-144.193,169.565,52.424,160.135
C04186=1014.418,299.471,-144.225,169.571,52.418,160.135
C04187=1014.424,299.719,-144.257,169.577,52.412,160.134
C04188=1014.430,299.967,-144.288,169.583,52.405,160.134
C04189=1014.436,300.215,-144.319,169.589,52.400,160.134
C04190=1014.442,300.463,-144.351,169.595,52.393,160.134
C04191=1014.447,300.711,-144.381,169.601,52.388,160.134
C04192=1014.453,300.959,-144.413,169.607,52.381,160.133
C04193=1014.460,301.206,-144.444,169.613,52.376,160.133
C04194=1014.466,301.454,-144.476,169.620,52.370,160.133
C04195=1014.471,301.702,-144.507,169.625,52.364,160.133
C04196=1014.477,301.950,-144.539,169.632,52.358,160.133
C04197=1014.484,302.198,-144.570,169.638,52.352,160.132
C04198=1014.489,302.446,-144.602,169.644,52.346,160.132
C04199=1014.496,302.694,-144.633,169.650,52.340,160.132
C04200=1014.501,302.942,-144.664,169.656,52.334,160.132
C04201=1014.508,303.190,-144.696,169.662,52.328,160.132
C04202=1014.514,303.438,-144.728,169.669,52.322,160.132
C04203=1014.519,303.685,-144.759,169.676,52.316,160.132
C04204=1014.526,303.933,-144.791,169.682,52.310,160.132
C04205=1014.532,304.181,-144.823,169.688,52.304,160.131
C04206=1014.538,304.429,-144.854,169.694,52.298,160.131
C04207=1014.544,304.677,-144.886,169.700,52.293,160.131
C04208=1014.551,304.925,-144.917,169.707,52.287,160.131
C04209=1014.556,305.172,-144.949,169.712,52.281,160.131
C04210=1014.563,305.420,-144.980,169.719,52.275,160.131
C04211=1014.569,305.668,-145.012,169.725,52.269,160.130
C04212=1014.576,305.916,-145.044,169.731,52.264,160.130
C04213=1014.581,306.164,-145.076,169.738,52.258,160.130
C04214=1014.588,306.412,-145.107,169.743,52.252,160.130
C04215=1014.594,306.660,-145.139,169.750,52.246,160.130
C04216=1014.601,306.908,-145.170,169.756,52.241,160.130
C04217=1014.607,307.156,-145.202,169.762,52.235,160.130
C04218=1014.612,307.404,-145.234,169.769,52.229,160.130
C04219=1014.620,307.683,-145.270,169.775,52.223,160.129
C04220=1014.627,307.962,-145.306,169.784,52.216,160.130
C04221=1014.634,308.241,-145.342,169.791,52.209,160.129
C04222=1014.641,308.520,-145.378,169.798,52.203,160.129
C04223=1014.647,308.768,-145.410,169.804,52.198,160.129
C04224=1014.653,309.015,-145.442,169.811,52.192,160.129
C04225=1014.660,309.263,-145.473,169.817,52.187,160.129
C04226=1014.666,309.511,-145.506,169.823,52.181,160.129
C04227=1014.671,309.759,-145.539,169.829,52.175,160.129
C04228=1014.678,310.007,-145.571,169.836,52.170,160.129
C04229=1014.684,310.255,-145.603,169.843,52.165,160.129
C04230=1014.689,310.502,-145.636,169.849,52.159,160.129
C04231=1014.696,310.750,-145.669,169.855,52.153,160.129
C04232=1014.702,310.997,-145.701,169.861,52.149,160.129
C04233=1014.707,311.246,-145.734,169.867,52.143,160.129
C04234=1014.714,311.493,-145.767,169.873,52.137,160.129
C04235=1014.720,311.741,-145.799,169.880,52.133,160.129
C04236=1014.726,311.988,-145.832,169.886,52.127,160.129
C04237=1014.732,312.237,-145.864,169.893,52.121,160.129
C04238=1014.738,312.484,-145.897,169.900,52.116,160.129
C04239=1014.744,312.732,-145.930,169.906,52.111,160.129
C04240=1014.750,312.980,-145.963,169.913,52.106,160.129
C04241=1014.757,313.227,-145.996,169.919,52.100,160.129
C04242=1014.763,313.476,-146.028,169.925,52.094,160.128
C04243=1014.769,313.723,-146.061,169.932,52.089,160.129
C04244=1014.774,313.971,-146.094,169.938,52.084,160.129
C04245=1014.781,314.219,-146.127,169.945,52.079,160.129
C04246=1014.787,314.466,-146.159,169.952,52.074,160.129
C04247=1014.793,314.714,-146.192,169.958,52.068,160.129
C04248=1014.800,314.961,-146.225,169.965,52.063,160.129
C04249=1014.805,315.209,-146.258,169.971,52.058,160.129
C04250=1014.811,315.457,-146.291,169.978,52.053,160.129
C04251=1014.818,315.705,-146.324,169.984,52.047,160.129
C04252=1014.824,315.952,-146.356,169.991,52.042,160.129
C04253=1014.830,316.200,-146.389,169.998,52.037,160.129
C04254=1014.837,316.448,-146.422,170.004,52.032,160.129
C04255=1014.843,316.696,-146.456,170.011,52.027,160.129
C04256=1014.849,316.943,-146.489,170.017,52.022,160.129
C04257=1014.856,317.190,-146.522,170.024,52.016,160.129
C04258=1014.862,317.438,-146.555,170.030,52.011,160.129
C04259=1014.869,317.686,-146.588,170.037,52.006,160.129
C04260=1014.874,317.934,-146.621,170.044,52.001,160.129
C04261=1014.881,318.182,-146.654,170.049,51.996,160.129
C04262=1014.887,318.429,-146.687,170.056,51.991,160.129
C04263=1014.894,318.677,-146.720,170.063,51.986,160.129
C04264=1014.900,318.925,-146.753,170.069,51.981,160.130
C04265=1014.906,319.173,-146.786,170.076,51.976,160.129
C04266=1014.913,319.420,-146.820,170.082,51.971,160.130
C04267=1014.919,319.668,-146.853,170.089,51.966,160.130
C04268=1014.926,319.916,-146.886,170.097,51.960,160.130
C04269=1014.932,320.162,-146.919,170.104,51.955,160.130
C04270=1014.939,320.411,-146.953,170.110,51.950,160.130
C04271=1014.945,320.659,-146.986,170.117,51.945,160.130
C04272=1014.952,320.906,-147.019,170.124,51.941,160.130
C04273=1014.958,321.154,-147.052,170.131,51.936,160.130
C04274=1014.964,321.401,-147.086,170.137,51.931,160.131
C04275=1014.971,321.650,-147.119,170.144,51.926,160.131
C04276=1014.978,321.896,-147.153,170.151,51.921,160.131
C04277=1014.985,322.145,-147.186,170.158,51.916,160.131
C04278=1014.991,322.392,-147.219,170.164,51.911,160.131
C04279=1014.999,322.676,-147.257,170.172,51.905,160.131
C04280=1015.006,322.962,-147.297,170.179,51.900,160.131
C04281=1015.013,323.247,-147.335,170.187,51.894,160.131
C04282=1015.021,323.531,-147.373,170.195,51.888,160.132
C04283=1015.028,323.779,-147.407,170.202,51.883,160.132
C04284=1015.035,324.026,-147.440,170.209,51.878,160.132
C04285=1015.041,324.274,-147.474,170.216,51.874,160.132
C04286=1015.047,324.521,-147.507,170.223,51.869,160.132
C04287=1015.055,324.769,-147.541,170.230,51.864,160.132
C04288=1015.061,325.017,-147.574,170.236,51.859,160.132
C04289=1015.068,325.264,-147.608,170.243,51.854,160.133
C04290=1015.075,325.512,-147.642,170.250,51.850,160.133
C04291=1015.081,325.759,-147.675,170.257,51.845,160.133
C04292=1015.088,326.007,-147.709,170.264,51.840,160.133
C04293=1015.094,326.254,-147.743,170.271,51.836,160.133
C04294=1015.101,326.502,-147.778,170.278,51.831,160.134
C04295=1015.108,326.750,-147.812,170.285,51.826,160.134
C04296=1015.114,326.997,-147.846,170.292,51.821,160.134
C04297=1015.120,327.245,-147.880,170.298,51.817,160.134
C04298=1015.127,327.493,-147.914,170.305,51.812,160.134
C04299=1015.133,327.740,-147.948,170.313,51.808,160.135
C04300=1015.140,327.988,-147.982,170.319,51.803,160.135
C04301=1015.147,328.236,-148.016,170.327,51.799,160.135
C04302=1015.153,328.482,-148.051,170.333,51.794,160.135
C04303=1015.160,328.730,-148.085,170.340,51.790,160.136
C04304=1015.167,328.978,-148.119,170.347,51.785,160.136
C04305=1015.173,329.226,-148.154,170.354,51.780,160.136
C04306=1015.179,329.473,-148.188,170.362,51.776,160.136
C04307=1015.187,329.720,-148.222,170.368,51.771,160.136
C04308=1015.193,329.968,-148.257,170.375,51.767,160.137
C04309=1015.200,330.216,-148.291,170.383,51.763,160.137
C04310=1015.206,330.463,-148.325,170.389,51.758,160.137
C04311=1015.213,330.711,-148.360,170.397,51.753,160.138
C04312=1015.220,330.958,-148.395,170.404,51.749,160.138
C04313=1015.227,331.206,-148.429,170.411,51.745,160.138
C04314=1015.233,331.454,-148.463,170.418,51.740,160.138
C04315=1015.240,331.701,-148.498,170.425,51.736,160.139
C04316=1015.247,331.949,-148.532,170.432,51.732,160.139
C04317=1015.254,332.195,-148.567,170.439,51.727,160.139
C04318=1015.260,332.443,-148.601,170.446,51.723,160.140
C04319=1015.267,332.691,-148.636,170.453,51.719,160.140
C04320=1015.274,332.938,-148.671,170.462,51.714,160.140
C04321=1015.280,333.186,-148.706,170.468,51.709,160.140
C04322=1015.287,333.433,-148.741,170.476,51.705,160.141
C04323=1015.294,333.680,-148.776,170.483,51.701,160.141
C04324=1015.301,333.928,-148.811,170.490,51.696,160.141
C04325=1015.307,334.176,-148.845,170.497,51.693,160.142
C04326=1015.314,334.423,-148.880,170.505,51.689,160.142
C04327=1015.321,334.671,-148.915,170.512,51.684,160.143
C04328=1015.328,334.918,-148.951,170.519,51.680,160.143
C04329=1015.335,335.165,-148.986,170.526,51.676,160.143
C04330=1015.341,335.413,-149.020,170.533,51.671,160.144
C04331=1015.348,335.661,-149.055,170.540,51.667,160.144
C04332=1015.355,335.908,-149.090,170.548,51.663,160.144
C04333=1015.361,336.155,-149.125,170.555,51.659,160.145
C04334=1015.368,336.403,-149.161,170.562,51.655,160.145
C04335=1015.375,336.650,-149.196,170.570,51.651,160.145
C04336=1015.382,336.897,-149.231,170.577,51.647,160.146
C04337=1015.389,337.146,-149.266,170.584,51.642,160.146
C04338=1015.396,337.393,-149.301,170.592,51.639,160.147
C04339=1015.404,337.673,-149.341,170.600,51.634,160.147
C04340=1015.412,337.954,-149.381,170.609,51.629,160.147
C04341=1015.419,338.233,-149.421,170.617,51.624,160.148
C04342=1015.427,338.514,-149.460,170.625,51.620,160.148
C04343=1015.435,338.762,-149.496,170.632,51.616,160.149
C04344=1015.441,339.009,-149.532,170.640,51.612,160.149
C04345=1015.448,339.256,-149.567,170.647,51.608,160.149
C04346=1015.455,339.504,-149.603,170.655,51.604,160.150
C04347=1015.462,339.750,-149.638,170.662,51.600,160.150
C04348=1015.469,339.998,-149.674,170.669,51.596,160.151
C04349=1015.476,340.246,-149.709,170.677,51.592,160.151
C04350=1015.482,340.493,-149.745,170.685,51.588,160.152
C04351=1015.490,340.741,-149.781,170.692,51.584,160.152
C04352=1015.497,340.988,-149.817,170.700,51.580,160.153
C04353=1015.503,341.235,-149.852,170.708,51.577,160.153
C04354=1015.511,341.483,-149.888,170.715,51.572,160.153
C04355=1015.517,341.730,-149.924,170.722,51.569,160.154
C04356=1015.524,341.977,-149.960,170.730,51.565,160.155
C04357=1015.532,342.225,-149.995,170.737,51.561,160.155
C04358=1015.539,342.472,-150.031,170.745,51.557,160.155
C04359=1015.546,342.718,-150.067,170.752,51.554,160.156
C04360=1015.552,342.967,-150.103,170.760,51.549,160.156
C04361=1015.559,343.214,-150.139,170.768,51.545,160.157
C04362=1015.567,343.461,-150.175,170.776,51.542,160.157
C04363=1015.573,343.709,-150.211,170.783,51.538,160.158
C04364=1015.581,343.956,-150.247,170.791,51.535,160.158
C04365=1015.588,344.203,-150.283,170.798,51.531,160.159
C04366=1015.596,344.450,-150.319,170.805,51.527,160.159
C04367=1015.602,344.698,-150.355,170.813,51.523,160.160
C04368=1015.609,344.945,-150.391,170.822,51.519,160.160
C04369=1015.616,345.192,-150.427,170.829,51.516,160.161
C04370=1015.623,345.440,-150.464,170.837,51.512,160.161
C04371=1015.630,345.687,-150.500,170.844,51.508,160.162
C04372=1015.638,345.934,-150.536,170.852,51.505,160.162
C04373=1015.645,346.181,-150.572,170.860,51.501,160.163
C04374=1015.652,346.429,-150.608,170.868,51.497,160.164
C04375=1015.660,346.676,-150.645,170.876,51.494,160.164
C04376=1015.666,346.923,-150.681,170.883,51.490,160.165
C04377=1015.674,347.171,-150.717,170.891,51.486,160.165
C04378=1015.681,347.417,-150.753,170.899,51.484,160.166
C04379=1015.688,347.665,-150.790,170.906,51.480,160.166
C04380=1015.696,347.912,-150.827,170.914,51.476,160.167
C04381=1015.702,348.159,-150.863,170.923,51.472,160.168
C04382=1015.710,348.406,-150.900,170.930,51.469,160.168
C04383=1015.717,348.654,-150.936,170.938,51.466,160.169
C04384=1015.724,348.901,-150.974,170.946,51.462,160.169
C04385=1015.731,349.148,-151.010,170.953,51.459,160.170
C04386=1015.738,349.396,-151.047,170.962,51.455,160.171
C04387=1015.746,349.643,-151.084,170.970,51.452,160.171
C04388=1015.753,349.890,-151.120,170.978,51.448,160.172
C04389=1015.760,350.137,-151.157,170.986,51.445,160.173
C04390=1015.767,350.384,-151.194,170.993,51.442,160.173
C04391=1015.775,350.631,-151.231,171.002,51.438,160.174
C04392=1015.782,350.879,-151.267,171.010,51.435,160.174
C04393=1015.790,351.126,-151.304,171.017,51.431,160.175
C04394=1015.796,351.373,-151.341,171.025,51.428,160.176
C04395=1015.804,351.620,-151.378,171.034,51.424,160.176
C04396=1015.811,351.867,-151.415,171.042,51.421,160.177
C04397=1015.819,352.114,-151.452,171.050,51.418,160.178
C04398=1015.827,352.361,-151.489,171.057,51.415,160.178
C04399=1015.834,352.631,-151.529,171.066,51.411,160.179
C04400=1015.842,352.899,-151.570,171.075,51.407,160.180
C04401=1015.851,353.168,-151.610,171.084,51.404,160.181
C04402=1015.858,353.437,-151.650,171.093,51.400,160.181
C04403=1015.866,353.684,-151.687,171.102,51.397,160.182
C04404=1015.874,353.931,-151.725,171.110,51.394,160.183
C04405=1015.881,354.178,-151.762,171.118,51.391,160.183
C04406=1015.888,354.425,-151.800,171.125,51.387,160.184
C04407=1015.896,354.672,-151.837,171.134,51.384,160.185
C04408=1015.903,354.919,-151.874,171.142,51.381,160.186
C04409=1015.911,355.167,-151.912,171.150,51.378,160.186
C04410=1015.919,355.413,-151.949,171.158,51.375,160.187
C04411=1015.926,355.660,-151.986,171.167,51.372,160.188
C04412=1015.933,355.908,-152.024,171.175,51.369,160.189
C04413=1015.940,356.155,-152.061,171.183,51.365,160.189
C04414=1015.948,356.402,-152.098,171.192,51.362,160.190
C04415=1015.956,356.649,-152.136,171.200,51.359,160.191
C04416=1015.964,356.896,-152.174,171.208,51.356,160.191
C04417=1015.971,357.143,-152.212,171.217,51.353,160.192
C04418=1015.978,357.390,-152.249,171.225,51.350,160.193
C04419=1015.986,357.637,-152.286,171.233,51.347,160.194
C04420=1015.994,357.884,-152.325,171.242,51.344,160.195
C04421=1016.002,358.131,-152.362,171.250,51.341,160.195
C04422=1016.009,358.379,-152.400,171.259,51.338,160.196
C04423=1016.016,358.625,-152.438,171.267,51.335,160.197
C04424=1016.025,358.873,-152.476,171.275,51.332,160.198
C04425=1016.033,359.119,-152.514,171.284,51.329,160.199
C04426=1016.040,359.366,-152.551,171.292,51.326,160.199
C04427=1016.047,359.613,-152.590,171.300,51.323,160.200
C04428=1016.055,359.861,-152.627,171.309,51.320,160.201
C04429=1016.062,360.107,-152.666,171.318,51.318,160.202
C04430=1016.070,360.354,-152.704,171.326,51.315,160.203
C04431=1016.077,360.602,-152.742,171.335,51.311,160.204
C04432=1016.085,360.848,-152.781,171.343,51.309,160.204
C04433=1016.092,361.095,-152.819,171.352,51.306,160.205
C04434=1016.101,361.342,-152.857,171.361,51.303,160.206
C04435=1016.109,361.598,-152.896,171.370,51.300,160.207
C04436=1016.116,361.853,-152.936,171.378,51.298,160.208
C04437=1016.125,362.109,-152.976,171.387,51.294,160.209
C04438=1016.132,362.365,-153.016,171.396,51.292,160.210
C04439=1016.140,362.612,-153.054,171.404,51.289,160.211
C04440=1016.148,362.859,-153.093,171.414,51.286,160.212
C04441=1016.156,363.106,-153.131,171.422,51.283,160.212
C04442=1016.163,363.352,-153.170,171.431,51.280,160.213
C04443=1016.172,363.600,-153.208,171.440,51.278,160.214
C04444=1016.179,363.846,-153.246,171.448,51.275,160.215
C04445=1016.187,364.093,-153.285,171.457,51.272,160.216
C04446=1016.195,364.340,-153.323,171.466,51.270,160.217
C04447=1016.203,364.587,-153.362,171.474,51.267,160.218
C04448=1016.211,364.834,-153.400,171.484,51.264,160.219
C04449=1016.219,365.080,-153.439,171.492,51.262,160.220
C04450=1016.226,365.328,-153.479,171.501,51.259,160.221
C04451=1016.235,365.575,-153.517,171.510,51.257,160.222
C04452=1016.242,365.822,-153.555,171.519,51.253,160.223
C04453=1016.250,366.069,-153.594,171.527,51.251,160.224
C04454=1016.259,366.315,-153.633,171.537,51.248,160.225
C04455=1016.266,366.562,-153.672,171.545,51.246,160.225
C04456=1016.274,366.809,-153.710,171.554,51.243,160.227
C04457=1016.283,367.056,-153.750,171.564,51.241,160.228
C04458=1016.291,367.303,-153.788,171.572,51.238,160.228
C04459=1016.300,367.588,-153.833,171.583,51.235,160.230
C04460=1016.309,367.873,-153.879,171.593,51.233,160.231
C04461=1016.318,368.158,-153.924,171.604,51.230,160.232
C04462=1016.327,368.443,-153.969,171.614,51.227,160.233
C04463=1016.335,368.690,-154.009,171.623,51.224,160.234
C04464=1016.343,368.937,-154.048,171.632,51.222,160.235
C04465=1016.352,369.184,-154.088,171.641,51.220,160.236
C04466=1016.359,369.431,-154.127,171.650,51.217,160.237
C04467=1016.367,369.677,-154.166,171.660,51.215,160.238
C04468=1016.375,369.924,-154.206,171.668,51.213,160.240
C04469=1016.383,370.170,-154.245,171.678,51.210,160.241
C04470=1016.392,370.417,-154.285,171.687,51.208,160.242
C04471=1016.400,370.664,-154.324,171.696,51.206,160.243
C04472=1016.408,370.911,-154.364,171.705,51.203,160.244
C04473=1016.416,371.157,-154.404,171.715,51.201,160.245
C04474=1016.424,371.404,-154.443,171.724,51.199,160.246
C04475=1016.433,371.651,-154.482,171.733,51.197,160.247
C04476=1016.440,371.898,-154.522,171.743,51.194,160.248
C04477=1016.449,372.144,-154.562,171.752,51.192,160.249
C04478=1016.457,372.391,-154.602,171.761,51.190,160.250
C04479=1016.465,372.638,-154.641,171.771,51.187,160.252
C04480=1016.473,372.884,-154.680,171.780,51.185,160.253
C04481=1016.482,373.131,-154.721,171.789,51.183,160.254
C04482=1016.491,373.378,-154.760,171.799,51.181,160.255
C04483=1016.498,373.625,-154.800,171.808,51.178,160.256
C04484=1016.507,373.871,-154.840,171.818,51.176,160.257
C04485=1016.516,374.117,-154.880,171.827,51.174,160.258
C04486=1016.523,374.364,-154.920,171.836,51.172,160.259
C04487=1016.533,374.611,-154.960,171.846,51.170,160.261
C04488=1016.540,374.858,-155.000,171.856,51.168,160.262
C04489=1016.549,375.104,-155.039,171.865,51.166,160.263
C04490=1016.558,375.350,-155.079,171.874,51.163,160.264
C04491=1016.566,375.598,-155.120,171.884,51.161,160.265
C04492=1016.574,375.844,-155.160,171.893,51.159,160.267
C04493=1016.583,376.090,-155.200,171.903,51.157,160.268
C04494=1016.591,376.337,-155.241,171.913,51.155,160.269
C04495=1016.599,376.584,-155.281,171.922,51.153,160.270
C04496=1016.607,376.830,-155.322,171.932,51.151,160.271
C04497=1016.616,377.077,-155.362,171.942,51.150,160.273
C04498=1016.624,377.323,-155.403,171.952,51.147,160.274
C04499=1016.632,377.570,-155.444,171.961,51.145,160.275
C04500=1016.641,377.817,-155.485,171.971,51.143,160.277
C04501=1016.650,378.063,-155.525,171.981,51.141,160.278
C04502=1016.658,378.309,-155.565,171.990,51.140,160.279
C04503=1016.666,378.556,-155.606,172.000,51.138,160.280
C04504=1016.675,378.802,-155.647,172.010,51.136,160.282
C04505=1016.684,379.049,-155.687,172.020,51.134,160.283
C04506=1016.692,379.295,-155.728,172.029,51.132,160.284
C04507=1016.701,379.542,-155.769,172.040,51.130,160.286
C04508=1016.709,379.788,-155.810,172.049,51.128,160.287
C04509=1016.718,380.035,-155.850,172.060,51.127,160.288
C04510=1016.727,380.281,-155.892,172.069,51.125,160.290
C04511=1016.735,380.528,-155.932,172.079,51.123,160.291
C04512=1016.744,380.774,-155.973,172.089,51.121,160.292
C04513=1016.752,381.021,-156.013,172.099,51.119,160.293
C04514=1016.761,381.267,-156.055,172.109,51.117,160.295
C04515=1016.770,381.514,-156.096,172.119,51.115,160.296
C04516=1016.779,381.759,-156.137,172.129,51.114,160.298
C04517=1016.788,382.006,-156.178,172.139,51.112,160.299
C04518=1016.796,382.253,-156.219,172.149,51.110,160.300
C04519=1016.807,382.561,-156.270,172.162,51.109,160.302
C04520=1016.819,382.868,-156.322,172.175,51.106,160.304
C04521=1016.829,383.176,-156.374,172.187,51.104,160.305
C04522=1016.841,383.484,-156.425,172.201,51.102,160.307
C04523=1016.849,383.731,-156.466,172.211,51.100,160.309
C04524=1016.858,383.977,-156.508,172.221,51.098,160.310
C04525=1016.868,384.223,-156.549,172.231,51.097,160.312
C04526=1016.877,384.470,-156.590,172.241,51.095,160.313
C04527=1016.886,384.717,-156.631,172.251,51.094,160.314
C04528=1016.894,384.962,-156.673,172.263,51.092,160.316
C04529=1016.903,385.209,-156.714,172.273,51.091,160.317
C04530=1016.912,385.455,-156.756,172.283,51.089,160.319
C04531=1016.921,385.701,-156.798,172.293,51.088,160.320
C04532=1016.930,385.948,-156.840,172.303,51.086,160.322
C04533=1016.939,386.194,-156.881,172.314,51.084,160.323
C04534=1016.948,386.440,-156.923,172.325,51.083,160.325
C04535=1016.957,386.686,-156.965,172.335,51.082,160.326
C04536=1016.966,386.932,-157.007,172.345,51.080,160.328
C04537=1016.975,387.179,-157.049,172.356,51.079,160.329
C04538=1016.984,387.425,-157.091,172.367,51.077,160.331
C04539=1016.993,387.671,-157.133,172.377,51.076,160.333
C04540=1017.002,387.918,-157.175,172.388,51.075,160.334
C04541=1017.011,388.164,-157.217,172.399,51.073,160.336
C04542=1017.020,388.410,-157.259,172.409,51.072,160.337
C04543=1017.029,388.657,-157.301,172.420,51.070,160.339
C04544=1017.039,388.902,-157.343,172.431,51.069,160.340
C04545=1017.047,389.149,-157.386,172.441,51.068,160.342
C04546=1017.057,389.395,-157.428,172.452,51.067,160.344
C04547=1017.066,389.641,-157.471,172.463,51.065,160.345
C04548=1017.075,389.887,-157.513,172.474,51.064,160.347
C04549=1017.084,390.133,-157.555,172.484,51.062,160.348
C04550=1017.094,390.380,-157.598,172.496,51.061,160.350
C04551=1017.103,390.626,-157.640,172.506,51.060,160.352
C04552=1017.111,390.872,-157.683,172.517,51.058,160.353
C04553=1017.121,391.119,-157.725,172.528,51.057,160.355
C04554=1017.130,391.364,-157.768,172.539,51.056,160.356
C04555=1017.140,391.610,-157.810,172.550,51.055,160.358
C04556=1017.150,391.856,-157.853,172.561,51.054,160.360
C04557=1017.159,392.102,-157.896,172.572,51.052,160.361
C04558=1017.168,392.349,-157.939,172.582,51.051,160.363
C04559=1017.177,392.595,-157.981,172.594,51.050,160.365
C04560=1017.187,392.841,-158.024,172.605,51.049,160.366
C04561=1017.195,393.087,-158.067,172.616,51.048,160.368
C04562=1017.205,393.334,-158.110,172.627,51.047,160.370
C04563=1017.215,393.579,-158.153,172.638,51.046,160.372
C04564=1017.224,393.826,-158.196,172.650,51.045,160.373
C04565=1017.233,394.071,-158.239,172.661,51.044,160.375
C04566=1017.243,394.318,-158.282,172.673,51.043,160.377
C04567=1017.252,394.563,-158.325,172.683,51.042,160.379
C04568=1017.262,394.810,-158.368,172.695,51.041,160.380
C04569=1017.272,395.055,-158.412,172.706,51.039,160.382
C04570=1017.280,395.301,-158.455,172.717,51.039,160.384
C04571=1017.290,395.547,-158.498,172.729,51.038,160.386
C04572=1017.300,395.794,-158.541,172.740,51.037,160.388
C04573=1017.309,396.039,-158.585,172.751,51.036,160.389
C04574=1017.319,396.285,-158.628,172.763,51.035,160.391
C04575=1017.329,396.531,-158.671,172.775,51.034,160.393
C04576=1017.339,396.778,-158.715,172.786,51.033,160.395
C04577=1017.349,397.023,-158.759,172.797,51.032,160.397
C04578=1017.358,397.269,-158.802,172.809,51.031,160.398
C04579=1017.375,397.680,-158.875,172.828,51.030,160.402
C04580=1017.390,398.089,-158.948,172.848,51.028,160.405
C04581=1017.406,398.499,-159.021,172.867,51.027,160.408
C04582=1017.423,398.910,-159.094,172.886,51.026,160.411
C04583=1017.432,399.156,-159.138,172.898,51.025,160.413
C04584=1017.442,399.400,-159.182,172.910,51.024,160.415
C04585=1017.452,399.646,-159.226,172.922,51.024,160.417
C04586=1017.462,399.893,-159.270,172.934,51.023,160.419
C04587=1017.472,400.139,-159.314,172.946,51.022,160.421
C04588=1017.482,400.384,-159.358,172.958,51.021,160.423
C04589=1017.492,400.630,-159.402,172.970,51.021,160.425
C04590=1017.501,400.876,-159.447,172.981,51.020,160.427
C04591=1017.511,401.122,-159.491,172.993,51.020,160.429
C04592=1017.521,401.367,-159.536,173.005,51.019,160.430
C04593=1017.531,401.613,-159.580,173.017,51.018,160.432
C04594=1017.540,401.859,-159.624,173.030,51.018,160.435
C04595=1017.551,402.105,-159.669,173.042,51.017,160.437
C04596=1017.561,402.351,-159.713,173.054,51.017,160.439
C04597=1017.571,402.597,-159.758,173.066,51.016,160.441
C04598=1017.580,402.842,-159.803,173.079,51.015,160.443
C04599=1017.591,403.088,-159.847,173.091,51.015,160.445
C04600=1017.601,403.333,-159.892,173.103,51.015,160.447
C04601=1017.611,403.579,-159.937,173.115,51.014,160.449
C04602=1017.622,403.825,-159.982,173.128,51.014,160.451
C04603=1017.632,404.070,-160.026,173.140,51.013,160.453
C04604=1017.641,404.316,-160.071,173.152,51.013,160.455
C04605=1017.652,404.562,-160.116,173.164,51.012,160.457
C04606=1017.662,404.807,-160.161,173.177,51.011,160.459
C04607=1017.672,405.054,-160.206,173.190,51.011,160.462
C04608=1017.682,405.299,-160.251,173.202,51.011,160.464
C04609=1017.693,405.545,-160.295,173.214,51.010,160.466
C04610=1017.703,405.790,-160.341,173.228,51.010,160.468
C04611=1017.713,406.036,-160.386,173.240,51.010,160.470
C04612=1017.723,406.282,-160.431,173.252,51.010,160.472
C04613=1017.735,406.527,-160.476,173.265,51.008,160.474
C04614=1017.745,406.773,-160.521,173.278,51.008,160.477
C04615=1017.755,407.019,-160.566,173.290,51.008,160.479
C04616=1017.766,407.264,-160.611,173.303,51.008,160.481
C04617=1017.776,407.510,-160.657,173.316,51.007,160.483
C04618=1017.787,407.756,-160.703,173.328,51.007,160.485
C04619=1017.797,408.001,-160.748,173.342,51.007,160.488
C04620=1017.808,408.246,-160.793,173.354,51.007,160.490
C04621=1017.819,408.492,-160.839,173.368,51.007,160.492
C04622=1017.829,408.738,-160.885,173.380,51.006,160.495
C04623=1017.840,408.984,-160.930,173.394,51.006,160.497
C04624=1017.850,409.229,-160.976,173.406,51.006,160.499
C04625=1017.861,409.475,-161.022,173.420,51.006,160.501
C04626=1017.871,409.721,-161.067,173.432,51.006,160.504
C04627=1017.881,409.966,-161.113,173.446,51.005,160.506
C04628=1017.892,410.210,-161.160,173.459,51.006,160.509
C04629=1017.903,410.456,-161.206,173.472,51.005,160.511
C04630=1017.914,410.702,-161.251,173.485,51.006,160.513
C04631=1017.549,408.705,-161.220,173.363,51.075,160.511
C04632=1017.539,408.459,-161.174,173.351,51.075,160.508
C04633=1017.529,408.215,-161.128,173.337,51.076,160.506
C04634=1017.518,407.968,-161.083,173.325,51.076,160.504
C04635=1017.508,407.723,-161.037,173.312,51.076,160.502
C04636=1017.497,407.477,-160.993,173.299,51.077,160.499
C04637=1017.486,407.231,-160.947,173.286,51.077,160.497
C04638=1017.476,406.986,-160.902,173.273,51.077,160.495
C04639=1017.465,406.740,-160.857,173.260,51.078,160.493
C04640=1017.455,406.494,-160.811,173.248,51.079,160.491
C04641=1017.445,406.249,-160.766,173.235,51.079,160.489
C04642=1017.434,406.003,-160.722,173.222,51.079,160.486
C04643=1017.424,405.758,-160.676,173.210,51.080,160.484
C04644=1017.414,405.512,-160.631,173.197,51.081,160.482
C04645=1017.403,405.266,-160.586,173.184,51.081,160.480
C04646=1017.393,405.020,-160.542,173.172,51.082,160.478
C04647=1017.383,404.775,-160.497,173.159,51.082,160.476
C04648=1017.373,404.529,-160.452,173.147,51.082,160.473
C04649=1017.362,404.283,-160.407,173.135,51.083,160.471
C04650=1017.352,404.037,-160.362,173.123,51.084,160.470
C04651=1017.342,403.792,-160.317,173.109,51.084,160.467
C04652=1017.333,403.546,-160.273,173.097,51.085,160.465
C04653=1017.321,403.300,-160.228,173.085,51.085,160.463
C04654=1017.312,403.055,-160.183,173.073,51.086,160.461
C04655=1017.302,402.809,-160.138,173.061,51.087,160.459
C04656=1017.291,402.563,-160.094,173.049,51.088,160.457
C04657=1017.282,402.317,-160.050,173.036,51.088,160.455
C04658=1017.272,402.072,-160.005,173.024,51.089,160.453
C04659=1017.261,401.826,-159.961,173.012,51.090,160.451
C04660=1017.252,401.580,-159.917,173.000,51.090,160.449
C04661=1017.242,401.335,-159.872,172.988,51.091,160.447
C04662=1017.232,401.089,-159.827,172.976,51.092,160.445
C04663=1017.222,400.843,-159.783,172.964,51.093,160.443
C04664=1017.212,400.597,-159.738,172.952,51.093,160.441
C04665=1017.203,400.351,-159.694,172.940,51.094,160.439
C04666=1017.193,400.105,-159.651,172.928,51.095,160.437
C04667=1017.183,399.860,-159.606,172.916,51.095,160.435
C04668=1017.173,399.614,-159.562,172.904,51.096,160.433
C04669=1017.163,399.368,-159.518,172.892,51.098,160.431
C04670=1017.154,399.122,-159.474,172.880,51.098,160.429
C04671=1017.144,398.876,-159.430,172.868,51.099,160.428
C04672=1017.129,398.496,-159.363,172.850,51.100,160.425
C04673=1017.114,398.115,-159.295,172.833,51.102,160.422
C04674=1017.099,397.736,-159.227,172.814,51.103,160.419
C04675=1017.084,397.356,-159.160,172.796,51.105,160.416
C04676=1017.074,397.110,-159.116,172.784,51.106,160.414
C04677=1017.065,396.864,-159.072,172.773,51.107,160.412
C04678=1017.055,396.617,-159.029,172.761,51.107,160.410
C04679=1017.045,396.371,-158.985,172.750,51.109,160.409
C04680=1017.036,396.126,-158.942,172.738,51.110,160.407
C04681=1017.026,395.880,-158.899,172.727,51.111,160.405
C04682=1017.017,395.633,-158.855,172.716,51.111,160.403
C04683=1017.007,395.387,-158.812,172.704,51.113,160.402
C04684=1016.997,395.142,-158.769,172.693,51.114,160.400
C04685=1016.988,394.895,-158.726,172.681,51.115,160.398
C04686=1016.979,394.650,-158.683,172.670,51.116,160.396
C04687=1016.969,394.403,-158.640,172.659,51.118,160.395
C04688=1016.959,394.157,-158.597,172.647,51.119,160.393
C04689=1016.950,393.912,-158.553,172.636,51.119,160.391
C04690=1016.940,393.665,-158.511,172.625,51.121,160.389
C04691=1016.931,393.419,-158.468,172.613,51.122,160.388
C04692=1016.922,393.173,-158.425,172.603,51.123,160.386
C04693=1016.913,392.927,-158.382,172.591,51.125,160.384
C04694=1016.902,392.681,-158.339,172.581,51.126,160.383
C04695=1016.894,392.435,-158.296,172.569,51.127,160.381
C04696=1016.884,392.189,-158.253,172.557,51.128,160.379
C04697=1016.875,391.943,-158.211,172.547,51.129,160.377
C04698=1016.866,391.697,-158.168,172.536,51.131,160.376
C04699=1016.857,391.450,-158.125,172.525,51.132,160.374
C04700=1016.848,391.204,-158.083,172.513,51.133,160.372
C04701=1016.838,390.958,-158.041,172.503,51.135,160.371
C04702=1016.829,390.712,-157.998,172.492,51.136,160.369
C04703=1016.819,390.466,-157.955,172.481,51.138,160.368
C04704=1016.810,390.220,-157.914,172.470,51.139,160.366
C04705=1016.800,389.973,-157.871,172.459,51.140,160.364
C04706=1016.792,389.727,-157.828,172.448,51.142,160.363
C04707=1016.783,389.481,-157.786,172.438,51.143,160.361
C04708=1016.774,389.235,-157.744,172.426,51.144,160.360
C04709=1016.764,388.988,-157.702,172.416,51.146,160.358
C04710=1016.755,388.742,-157.659,172.406,51.147,160.356
C04711=1016.746,388.496,-157.617,172.394,51.149,160.355
C04712=1016.737,388.250,-157.575,172.384,51.150,160.353
C04713=1016.729,388.003,-157.533,172.373,51.152,160.352
C04714=1016.719,387.758,-157.490,172.362,51.153,160.350
C04715=1016.710,387.511,-157.449,172.352,51.155,160.349
C04716=1016.702,387.265,-157.407,172.341,51.156,160.347
C04717=1016.693,387.019,-157.365,172.331,51.158,160.346
C04718=1016.684,386.772,-157.323,172.321,51.159,160.344
C04719=1016.674,386.527,-157.281,172.309,51.161,160.343
C04720=1016.666,386.280,-157.239,172.299,51.162,160.341
C04721=1016.657,386.034,-157.198,172.289,51.164,160.340
C04722=1016.648,385.787,-157.156,172.277,51.166,160.338
C04723=1016.639,385.541,-157.114,172.268,51.168,160.337
C04724=1016.630,385.295,-157.072,172.257,51.169,160.335
C04725=1016.621,385.048,-157.031,172.247,51.171,160.334
C04726=1016.612,384.802,-156.989,172.236,51.173,160.332
C04727=1016.603,384.555,-156.949,172.226,51.174,160.331
C04728=1016.594,384.309,-156.907,172.216,51.176,160.330
C04729=1016.585,384.063,-156.865,172.205,51.177,160.328
C04730=1016.576,383.816,-156.823,172.195,51.180,160.327
C04731=1016.567,383.570,-156.783,172.184,51.181,160.325
C04732=1016.556,383.260,-156.731,172.172,51.183,160.324
C04733=1016.545,382.950,-156.680,172.159,51.185,160.322
C04734=1016.533,382.639,-156.627,172.147,51.188,160.320
C04735=1016.522,382.330,-156.576,172.133,51.190,160.318
C04736=1016.513,382.083,-156.535,172.123,51.192,160.317
C04737=1016.505,381.837,-156.493,172.113,51.194,160.316
C04738=1016.496,381.590,-156.453,172.103,51.195,160.314
C04739=1016.487,381.343,-156.412,172.093,51.197,160.313
C04740=1016.479,381.098,-156.371,172.083,51.200,160.312
C04741=1016.470,380.851,-156.330,172.072,51.201,160.310
C04742=1016.461,380.605,-156.290,172.063,51.204,160.309
C04743=1016.452,380.358,-156.248,172.052,51.205,160.307
C04744=1016.444,380.111,-156.207,172.043,51.207,160.306
C04745=1016.435,379.865,-156.167,172.033,51.209,160.305
C04746=1016.426,379.619,-156.126,172.023,51.211,160.304
C04747=1016.418,379.372,-156.085,172.013,51.213,160.302
C04748=1016.410,379.125,-156.044,172.003,51.215,160.301
C04749=1016.401,378.879,-156.004,171.993,51.217,160.300
C04750=1016.392,378.632,-155.963,171.983,51.219,160.299
C04751=1016.384,378.386,-155.922,171.974,51.221,160.297
C04752=1016.376,378.139,-155.881,171.964,51.223,160.296
C04753=1016.367,377.893,-155.841,171.954,51.225,160.295
C04754=1016.359,377.647,-155.801,171.944,51.227,160.293
C04755=1016.350,377.400,-155.760,171.934,51.229,160.292
C04756=1016.342,377.153,-155.719,171.924,51.231,160.291
C04757=1016.334,376.908,-155.679,171.914,51.233,160.290
C04758=1016.325,376.660,-155.639,171.905,51.235,160.288
C04759=1016.317,376.414,-155.598,171.895,51.237,160.287
C04760=1016.309,376.167,-155.558,171.886,51.240,160.286
C04761=1016.300,375.921,-155.518,171.877,51.242,160.285
C04762=1016.292,375.674,-155.477,171.867,51.244,160.284
C04763=1016.284,375.427,-155.437,171.857,51.246,160.282
C04764=1016.276,375.181,-155.397,171.847,51.248,160.281
C04765=1016.267,374.935,-155.357,171.838,51.251,160.280
C04766=1016.259,374.687,-155.317,171.828,51.253,160.279
C04767=1016.250,374.441,-155.277,171.818,51.255,160.278
C04768=1016.242,374.194,-155.237,171.810,51.257,160.277
C04769=1016.234,373.948,-155.198,171.800,51.259,160.276
C04770=1016.225,373.701,-155.158,171.790,51.262,160.274
C04771=1016.216,373.454,-155.117,171.781,51.264,160.273
C04772=1016.208,373.208,-155.078,171.771,51.266,160.272
C04773=1016.200,372.961,-155.038,171.762,51.269,160.271
C04774=1016.192,372.714,-154.999,171.752,51.271,160.270
C04775=1016.183,372.468,-154.959,171.744,51.274,160.269
C04776=1016.175,372.221,-154.919,171.734,51.276,160.268
C04777=1016.167,371.975,-154.879,171.724,51.278,160.267
C04778=1016.159,371.728,-154.840,171.715,51.281,160.266
C04779=1016.151,371.481,-154.800,171.706,51.283,160.264
C04780=1016.142,371.235,-154.761,171.697,51.286,160.263
C04781=1016.135,370.988,-154.721,171.687,51.288,160.262
C04782=1016.126,370.741,-154.682,171.678,51.290,160.261
C04783=1016.118,370.494,-154.642,171.669,51.293,160.260
C04784=1016.110,370.247,-154.603,171.660,51.295,160.259
C04785=1016.102,370.000,-154.564,171.650,51.298,160.258
C04786=1016.094,369.753,-154.524,171.641,51.300,160.257
C04787=1016.086,369.507,-154.485,171.632,51.303,160.256
C04788=1016.078,369.261,-154.445,171.623,51.305,160.255
C04789=1016.070,369.013,-154.406,171.613,51.308,160.254
C04790=1016.062,368.767,-154.367,171.605,51.310,160.253
C04791=1016.054,368.520,-154.327,171.596,51.313,160.252
C04792=1016.045,368.232,-154.282,171.585,51.315,160.250
C04793=1016.035,367.945,-154.236,171.574,51.319,160.249
C04794=1016.026,367.657,-154.191,171.564,51.322,160.248
C04795=1016.017,367.370,-154.145,171.554,51.325,160.247
C04796=1016.010,367.123,-154.105,171.544,51.327,160.246
C04797=1016.001,366.876,-154.067,171.535,51.330,160.245
C04798=1015.993,366.629,-154.028,171.526,51.332,160.244
C04799=1015.985,366.383,-153.989,171.517,51.335,160.243
C04800=1015.977,366.136,-153.951,171.508,51.338,160.242
C04801=1015.969,365.889,-153.912,171.500,51.341,160.241
C04802=1015.962,365.642,-153.874,171.490,51.344,160.240
C04803=1015.953,365.395,-153.834,171.482,51.346,160.239
C04804=1015.945,365.148,-153.796,171.473,51.349,160.238
C04805=1015.937,364.902,-153.758,171.464,51.352,160.237
C04806=1015.929,364.655,-153.719,171.455,51.354,160.236
C04807=1015.921,364.407,-153.680,171.446,51.358,160.236
C04808=1015.914,364.161,-153.642,171.438,51.360,160.235
C04809=1015.905,363.914,-153.604,171.429,51.363,160.234
C04810=1015.898,363.667,-153.565,171.419,51.366,160.233
C04811=1015.891,363.420,-153.526,171.411,51.368,160.232
C04812=1015.883,363.173,-153.488,171.402,51.372,160.231
C04813=1015.875,362.926,-153.449,171.394,51.374,160.230
C04814=1015.867,362.679,-153.411,171.385,51.377,160.229
C04815=1015.859,362.432,-153.372,171.376,51.380,160.228
C04816=1015.852,362.186,-153.334,171.367,51.383,160.228
C04817=1015.843,361.938,-153.296,171.359,51.386,160.227
C04818=1015.836,361.691,-153.258,171.350,51.389,160.226
C04819=1015.829,361.445,-153.220,171.342,51.392,160.225
C04820=1015.820,361.197,-153.181,171.333,51.395,160.224
C04821=1015.813,360.951,-153.143,171.324,51.397,160.223
C04822=1015.806,360.704,-153.105,171.315,51.401,160.222
C04823=1015.798,360.457,-153.067,171.307,51.404,160.222
C04824=1015.790,360.210,-153.029,171.298,51.406,160.221
C04825=1015.783,359.963,-152.991,171.290,51.409,160.220
C04826=1015.775,359.716,-152.952,171.282,51.412,160.219
C04827=1015.768,359.469,-152.914,171.273,51.416,160.218
C04828=1015.761,359.222,-152.876,171.265,51.419,160.218
C04829=1015.753,358.975,-152.838,171.256,51.421,160.217
C04830=1015.744,358.728,-152.800,171.248,51.424,160.216
C04831=1015.737,358.481,-152.763,171.239,51.428,160.215
C04832=1015.730,358.234,-152.725,171.231,51.431,160.214
C04833=1015.722,357.987,-152.687,171.222,51.434,160.213
C04834=1015.715,357.739,-152.649,171.214,51.437,160.213
C04835=1015.706,357.493,-152.612,171.206,51.440,160.212
C04836=1015.699,357.246,-152.574,171.197,51.443,160.211
C04837=1015.692,356.999,-152.537,171.189,51.446,160.210
C04838=1015.684,356.752,-152.499,171.180,51.449,160.210
C04839=1015.677,356.504,-152.462,171.172,51.453,160.209
C04840=1015.669,356.258,-152.425,171.163,51.456,160.208
C04841=1015.661,356.010,-152.387,171.155,51.459,160.208
C04842=1015.654,355.763,-152.348,171.147,51.462,160.207
C04843=1015.647,355.516,-152.311,171.138,51.466,160.206
C04844=1015.639,355.269,-152.274,171.131,51.469,160.205
C04845=1015.631,355.022,-152.236,171.123,51.472,160.205
C04846=1015.624,354.775,-152.199,171.114,51.476,160.204
C04847=1015.616,354.528,-152.163,171.106,51.479,160.203
C04848=1015.609,354.280,-152.125,171.097,51.483,160.203
C04849=1015.602,354.033,-152.088,171.089,51.485,160.202
C04850=1015.595,353.786,-152.050,171.081,51.488,160.201
C04851=1015.587,353.539,-152.013,171.073,51.492,160.200
C04852=1015.579,353.260,-151.971,171.064,51.496,160.200
C04853=1015.571,352.980,-151.929,171.054,51.500,160.199
C04854=1015.562,352.699,-151.887,171.045,51.503,160.198
C04855=1015.554,352.420,-151.845,171.036,51.507,160.197
C04856=1015.546,352.173,-151.809,171.027,51.511,160.197
C04857=1015.539,351.925,-151.771,171.020,51.514,160.196
C04858=1015.531,351.679,-151.735,171.012,51.518,160.196
C04859=1015.524,351.431,-151.698,171.003,51.521,160.195
C04860=1015.517,351.184,-151.660,170.996,51.525,160.194
C04861=1015.510,350.937,-151.624,170.988,51.528,160.193
C04862=1015.502,350.690,-151.587,170.979,51.532,160.193
C04863=1015.495,350.442,-151.551,170.972,51.535,160.192
C04864=1015.487,350.195,-151.513,170.964,51.538,160.192
C04865=1015.480,349.948,-151.477,170.955,51.542,160.191
C04866=1015.473,349.701,-151.440,170.947,51.546,160.190
C04867=1015.465,349.454,-151.403,170.940,51.550,160.190
C04868=1015.459,349.206,-151.367,170.932,51.553,160.189
C04869=1015.451,348.959,-151.331,170.923,51.557,160.189
C04870=1015.444,348.712,-151.293,170.916,51.560,160.188
C04871=1015.437,348.465,-151.257,170.908,51.564,160.187
C04872=1015.430,348.218,-151.221,170.901,51.567,160.187
C04873=1015.423,347.970,-151.184,170.892,51.571,160.186
C04874=1015.415,347.723,-151.147,170.884,51.574,160.186
C04875=1015.409,347.476,-151.110,170.876,51.578,160.185
C04876=1015.401,347.229,-151.074,170.869,51.582,160.185
C04877=1015.394,346.981,-151.038,170.860,51.586,160.184
C04878=1015.387,346.734,-151.002,170.853,51.589,160.183
C04879=1015.380,346.487,-150.965,170.845,51.593,160.183
C04880=1015.373,346.240,-150.929,170.837,51.596,160.182
C04881=1015.366,345.992,-150.893,170.829,51.600,160.182
C04882=1015.359,345.746,-150.857,170.822,51.605,160.181
C04883=1015.351,345.498,-150.821,170.814,51.608,160.181
C04884=1015.344,345.250,-150.784,170.807,51.612,160.180
C04885=1015.337,345.003,-150.749,170.798,51.616,160.180
C04886=1015.329,344.756,-150.712,170.790,51.620,160.179
C04887=1015.323,344.508,-150.676,170.783,51.623,160.179
C04888=1015.315,344.261,-150.640,170.776,51.627,160.178
C04889=1015.309,344.014,-150.605,170.767,51.631,160.178
C04890=1015.302,343.767,-150.569,170.759,51.635,160.177
C04891=1015.295,343.519,-150.532,170.752,51.639,160.177
C04892=1015.288,343.272,-150.496,170.745,51.643,160.176
C04893=1015.280,343.024,-150.461,170.737,51.646,160.176
C04894=1015.274,342.777,-150.424,170.729,51.650,160.175
C04895=1015.267,342.530,-150.389,170.721,51.655,160.175
C04896=1015.259,342.282,-150.353,170.714,51.658,160.174
C04897=1015.252,342.036,-150.317,170.706,51.662,160.174
C04898=1015.245,341.788,-150.281,170.699,51.666,160.173
C04899=1015.239,341.541,-150.245,170.692,51.670,160.173
C04900=1015.232,341.293,-150.210,170.683,51.674,160.173
C04901=1015.225,341.046,-150.175,170.676,51.678,160.172
C04902=1015.217,340.798,-150.139,170.669,51.682,160.172
C04903=1015.211,340.551,-150.103,170.661,51.686,160.171
C04904=1015.204,340.304,-150.067,170.654,51.690,160.171
C04905=1015.197,340.056,-150.031,170.646,51.694,160.170
C04906=1015.190,339.809,-149.996,170.638,51.698,160.170
C04907=1015.183,339.562,-149.960,170.631,51.703,160.170
C04908=1015.176,339.314,-149.925,170.623,51.706,160.169
C04909=1015.170,339.067,-149.890,170.616,51.711,160.169
C04910=1015.163,338.819,-149.854,170.609,51.714,160.168
C04911=1015.156,338.572,-149.818,170.601,51.719,160.168
C04912=1015.148,338.290,-149.778,170.592,51.724,160.167
C04913=1015.140,338.007,-149.739,170.584,51.728,160.167
C04914=1015.132,337.724,-149.698,170.576,51.733,160.166
C04915=1015.125,337.442,-149.658,170.567,51.738,160.166
C04916=1015.118,337.194,-149.623,170.560,51.742,160.166
C04917=1015.110,336.946,-149.587,170.553,51.746,160.165
C04918=1015.104,336.699,-149.552,170.545,51.751,160.165
C04919=1015.097,336.452,-149.517,170.538,51.755,160.165
C04920=1015.090,336.204,-149.482,170.531,51.759,160.164
C04921=1015.083,335.957,-149.447,170.523,51.764,160.164
C04922=1015.077,335.709,-149.412,170.515,51.767,160.163
C04923=1015.069,335.462,-149.378,170.508,51.772,160.163
C04924=1015.063,335.214,-149.343,170.501,51.776,160.163
C04925=1015.056,334.967,-149.308,170.494,51.780,160.162
C04926=1015.049,334.720,-149.273,170.487,51.785,160.162
C04927=1015.042,334.472,-149.237,170.479,51.789,160.162
C04928=1015.036,334.224,-149.203,170.472,51.793,160.161
C04929=1015.029,333.977,-149.168,170.465,51.798,160.161
C04930=1015.022,333.730,-149.133,170.457,51.803,160.161
C04931=1015.016,333.482,-149.098,170.450,51.807,160.161
C04932=1015.009,333.234,-149.063,170.443,51.811,160.160
C04933=1015.002,332.987,-149.028,170.436,51.816,160.160
C04934=1014.996,332.740,-148.994,170.429,51.820,160.160
C04935=1014.990,332.492,-148.959,170.422,51.824,160.159
C04936=1014.982,332.245,-148.924,170.414,51.828,160.159
C04937=1014.976,331.997,-148.890,170.408,51.833,160.159
C04938=1014.969,331.749,-148.855,170.400,51.838,160.158
C04939=1014.962,331.502,-148.820,170.392,51.842,160.158
C04940=1014.955,331.254,-148.787,170.386,51.847,160.158
C04941=1014.949,331.008,-148.752,170.378,51.851,160.158
C04942=1014.943,330.760,-148.717,170.371,51.856,160.157
C04943=1014.935,330.512,-148.683,170.365,51.861,160.157
C04944=1014.929,330.264,-148.648,170.357,51.865,160.157
C04945=1014.922,330.017,-148.614,170.350,51.869,160.157
C04946=1014.916,329.770,-148.580,170.344,51.874,160.157
C04947=1014.909,329.522,-148.546,170.335,51.879,160.156
C04948=1014.902,329.274,-148.511,170.329,51.884,160.156
C04949=1014.895,329.027,-148.477,170.321,51.888,160.156
C04950=1014.889,328.779,-148.443,170.315,51.893,160.156
C04951=1014.883,328.531,-148.409,170.308,51.897,160.155
C04952=1014.876,328.284,-148.375,170.301,51.902,160.155
C04953=1014.870,328.036,-148.341,170.294,51.907,160.155
C04954=1014.863,327.789,-148.306,170.287,51.911,160.155
C04955=1014.856,327.541,-148.272,170.280,51.916,160.154
C04956=1014.850,327.294,-148.238,170.273,51.921,160.154
C04957=1014.844,327.046,-148.203,170.266,51.926,160.154
C04958=1014.837,326.799,-148.170,170.259,51.930,160.154
C04959=1014.830,326.551,-148.135,170.251,51.935,160.154
C04960=1014.824,326.303,-148.101,170.245,51.940,160.153
C04961=1014.817,326.056,-148.068,170.237,51.944,160.153
C04962=1014.811,325.808,-148.033,170.231,51.949,160.153
C04963=1014.804,325.561,-148.000,170.224,51.954,160.153
C04964=1014.797,325.313,-147.967,170.217,51.959,160.153
C04965=1014.791,325.066,-147.933,170.210,51.964,160.152
C04966=1014.784,324.818,-147.899,170.203,51.969,160.152
C04967=1014.777,324.570,-147.866,170.197,51.974,160.152
C04968=1014.771,324.323,-147.832,170.189,51.979,160.152
C04969=1014.764,324.074,-147.799,170.182,51.984,160.152
C04970=1014.757,323.827,-147.766,170.175,51.989,160.152
C04971=1014.751,323.579,-147.731,170.169,51.994,160.152
C04972=1014.743,323.292,-147.692,170.161,51.999,160.151
C04973=1014.736,323.005,-147.654,170.153,52.005,160.151
C04974=1014.728,322.719,-147.615,170.145,52.011,160.151
C04975=1014.721,322.432,-147.577,170.137,52.017,160.151
C04976=1014.714,322.184,-147.543,170.130,52.022,160.151
C04977=1014.708,321.937,-147.510,170.123,52.027,160.151
C04978=1014.701,321.689,-147.477,170.116,52.032,160.151
C04979=1014.694,321.442,-147.443,170.110,52.037,160.151
C04980=1014.688,321.194,-147.410,170.103,52.042,160.150
C04981=1014.682,320.946,-147.377,170.097,52.048,160.151
C04982=1014.675,320.699,-147.344,170.090,52.052,160.150
C04983=1014.668,320.450,-147.310,170.083,52.057,160.150
C04984=1014.662,320.203,-147.278,170.076,52.062,160.150
C04985=1014.656,319.955,-147.244,170.069,52.068,160.150
C04986=1014.650,319.708,-147.211,170.062,52.073,160.150
C04987=1014.643,319.460,-147.178,170.056,52.078,160.150
C04988=1014.636,319.212,-147.145,170.049,52.083,160.150
C04989=1014.630,318.965,-147.112,170.042,52.088,160.150
C04990=1014.624,318.716,-147.078,170.036,52.093,160.150
C04991=1014.617,318.469,-147.045,170.029,52.099,160.150
C04992=1014.611,318.221,-147.012,170.022,52.104,160.150
C04993=1014.605,317.974,-146.980,170.016,52.109,160.149
C04994=1014.598,317.727,-146.946,170.009,52.114,160.150
C04995=1014.592,317.478,-146.913,170.003,52.119,160.149
C04996=1014.586,317.230,-146.880,169.996,52.124,160.149
C04997=1014.579,316.983,-146.847,169.989,52.130,160.149
C04998=1014.573,316.735,-146.814,169.982,52.135,160.149
C04999=1014.567,316.488,-146.782,169.976,52.141,160.149
C05000=1014.561,316.240,-146.748,169.969,52.146,160.149
C05001=1014.554,315.991,-146.715,169.963,52.152,160.149
C05002=1014.548,315.744,-146.682,169.956,52.157,160.149
C05003=1014.542,315.496,-146.650,169.950,52.162,160.149
C05004=1014.536,315.249,-146.617,169.943,52.167,160.149
C05005=1014.530,315.001,-146.584,169.937,52.173,160.149
C05006=1014.524,314.753,-146.551,169.930,52.178,160.149
C05007=1014.517,314.506,-146.518,169.924,52.183,160.149
C05008=1014.511,314.258,-146.485,169.917,52.188,160.149
C05009=1014.505,314.010,-146.453,169.911,52.194,160.149
C05010=1014.499,313.763,-146.420,169.904,52.199,160.149
C05011=1014.493,313.514,-146.387,169.898,52.205,160.149
C05012=1014.487,313.267,-146.354,169.891,52.210,160.149
C05013=1014.481,313.019,-146.322,169.885,52.215,160.149
C05014=1014.474,312.771,-146.289,169.878,52.221,160.149
C05015=1014.468,312.524,-146.256,169.872,52.227,160.149
C05016=1014.463,312.275,-146.224,169.865,52.232,160.149
C05017=1014.457,312.028,-146.191,169.859,52.237,160.149
C05018=1014.451,311.781,-146.158,169.853,52.243,160.149
C05019=1014.445,311.533,-146.126,169.845,52.248,160.149
C05020=1014.439,311.285,-146.094,169.839,52.254,160.149
C05021=1014.432,311.037,-146.061,169.832,52.260,160.149
C05022=1014.427,310.790,-146.028,169.826,52.265,160.149
C05023=1014.421,310.541,-145.996,169.819,52.270,160.149
C05024=1014.415,310.294,-145.963,169.813,52.276,160.149
C05025=1014.409,310.046,-145.931,169.807,52.282,160.149
C05026=1014.403,309.799,-145.898,169.800,52.287,160.149
C05027=1014.397,309.551,-145.866,169.794,52.293,160.149
C05028=1014.391,309.303,-145.833,169.788,52.298,160.150
C05029=1014.384,309.055,-145.801,169.782,52.304,160.150
C05030=1014.379,308.808,-145.769,169.775,52.310,160.150
C05031=1014.372,308.560,-145.738,169.769,52.315,160.150
C05032=1014.365,308.279,-145.701,169.762,52.322,160.150
C05033=1014.358,307.997,-145.665,169.754,52.329,160.150
C05034=1014.351,307.715,-145.629,169.747,52.335,160.150
C05035=1014.344,307.434,-145.593,169.740,52.342,160.150
C05036=1014.338,307.186,-145.561,169.734,52.348,160.150
C05037=1014.332,306.938,-145.529,169.728,52.353,160.151
C05038=1014.325,306.690,-145.498,169.721,52.359,160.151
C05039=1014.319,306.443,-145.466,169.714,52.365,160.151
C05040=1014.313,306.195,-145.435,169.708,52.371,160.151
C05041=1014.307,305.947,-145.403,169.702,52.377,160.151
C05042=1014.300,305.699,-145.371,169.696,52.383,160.151
C05043=1014.295,305.451,-145.340,169.689,52.388,160.151
C05044=1014.289,305.203,-145.308,169.683,52.395,160.151
C05045=1014.282,304.955,-145.276,169.677,52.400,160.152
C05046=1014.276,304.708,-145.245,169.670,52.406,160.152
C05047=1014.270,304.460,-145.213,169.664,52.413,160.152
C05048=1014.264,304.211,-145.181,169.658,52.418,160.152
C05049=1014.258,303.964,-145.150,169.651,52.424,160.152
C05050=1014.252,303.716,-145.118,169.646,52.430,160.152
C05051=1014.245,303.468,-145.087,169.639,52.436,160.152
C05052=1014.240,303.220,-145.056,169.633,52.443,160.153
C05053=1014.233,302.972,-145.024,169.627,52.448,160.153
C05054=1014.228,302.725,-144.993,169.620,52.455,160.153
C05055=1014.221,302.477,-144.961,169.614,52.461,160.153
C05056=1014.215,302.228,-144.930,169.608,52.466,160.153
C05057=1014.209,301.981,-144.899,169.602,52.473,160.153
C05058=1014.203,301.732,-144.867,169.596,52.478,160.154
C05059=1014.197,301.485,-144.836,169.590,52.485,160.154
C05060=1014.191,301.236,-144.804,169.584,52.490,160.154
C05061=1014.186,300.989,-144.773,169.578,52.497,160.154
C05062=1014.179,300.741,-144.741,169.571,52.503,160.154
C05063=1014.174,300.493,-144.710,169.565,52.509,160.155
C05064=1014.168,300.245,-144.679,169.559,52.516,160.155
C05065=1014.162,299.997,-144.648,169.552,52.521,160.155
C05066=1014.156,299.749,-144.617,169.547,52.528,160.155
C05067=1014.150,299.501,-144.585,169.541,52.534,160.156
C05068=1014.145,299.254,-144.555,169.535,52.540,160.156
C05069=1014.139,299.005,-144.523,169.529,52.546,160.156
C05070=1014.133,298.758,-144.492,169.522,52.553,160.156
C05071=1014.127,298.509,-144.460,169.516,52.558,160.156
C05072=1014.121,298.262,-144.430,169.510,52.565,160.156
C05073=1014.116,298.014,-144.398,169.504,52.571,160.157
C05074=1014.109,297.765,-144.367,169.498,52.577,160.157
C05075=1014.104,297.518,-144.336,169.492,52.583,160.157
C05076=1014.097,297.269,-144.305,169.486,52.590,160.157
C05077=1014.092,297.022,-144.273,169.480,52.596,160.158
C05078=1014.086,296.774,-144.243,169.474,52.602,160.158
C05079=1014.081,296.526,-144.212,169.467,52.608,160.158
C05080=1014.074,296.278,-144.181,169.461,52.615,160.158
C05081=1014.069,296.030,-144.150,169.455,52.621,160.159
C05082=1014.063,295.782,-144.119,169.450,52.628,160.159
C05083=1014.057,295.534,-144.087,169.444,52.634,160.159
C05084=1014.052,295.286,-144.056,169.438,52.640,160.160
C05085=1014.047,295.038,-144.026,169.432,52.646,160.160
C05086=1014.041,294.790,-143.994,169.426,52.652,160.160
C05087=1014.035,294.542,-143.964,169.420,52.659,160.160
C05088=1014.030,294.294,-143.933,169.413,52.666,160.160
C05089=1014.024,294.046,-143.902,169.407,52.672,160.161
C05090=1014.018,293.798,-143.871,169.402,52.678,160.161
C05091=1014.013,293.551,-143.840,169.396,52.685,160.161
C05092=1014.006,293.287,-143.807,169.389,52.692,160.161
C05093=1014.001,293.023,-143.774,169.384,52.699,160.162
C05094=1013.994,292.760,-143.742,169.377,52.705,160.162
C05095=1013.988,292.497,-143.709,169.371,52.712,160.162
C05096=1013.982,292.249,-143.679,169.364,52.719,160.163
C05097=1013.977,292.001,-143.648,169.359,52.726,160.163
C05098=1013.972,291.753,-143.617,169.353,52.732,160.163
C05099=1013.966,291.505,-143.587,169.347,52.738,160.164
C05100=1013.960,291.257,-143.557,169.341,52.745,160.164
C05101=1013.954,291.009,-143.527,169.335,52.751,160.164
C05102=1013.949,290.761,-143.497,169.329,52.759,160.165
C05103=1013.942,290.512,-143.466,169.323,52.765,160.165
C05104=1013.936,290.265,-143.436,169.317,52.771,160.165
C05105=1013.931,290.017,-143.405,169.312,52.778,160.166
C05106=1013.925,289.768,-143.376,169.306,52.785,160.166
C05107=1013.919,289.520,-143.345,169.299,52.792,160.166
C05108=1013.913,289.273,-143.315,169.294,52.799,160.167
C05109=1013.908,289.025,-143.285,169.288,52.805,160.167
C05110=1013.903,288.776,-143.254,169.282,52.812,160.167
C05111=1013.897,288.528,-143.224,169.276,52.819,160.168
C05112=1013.892,288.280,-143.194,169.270,52.825,160.168
C05113=1013.886,288.032,-143.164,169.265,52.833,160.169
C05114=1013.880,287.784,-143.134,169.259,52.839,160.169
C05115=1013.874,287.536,-143.104,169.253,52.845,160.169
C05116=1013.869,287.288,-143.074,169.247,52.853,160.170
C05117=1013.863,287.039,-143.044,169.241,52.859,160.170
C05118=1013.857,286.792,-143.014,169.236,52.866,160.170
C05119=1013.852,286.543,-142.984,169.230,52.873,160.171
C05120=1013.846,286.295,-142.954,169.224,52.880,160.171
C05121=1013.840,286.047,-142.924,169.218,52.887,160.171
C05122=1013.835,285.799,-142.894,169.212,52.894,160.172
C05123=1013.828,285.551,-142.865,169.207,52.901,160.172
C05124=1013.822,285.303,-142.834,169.200,52.908,160.173
C05125=1013.817,285.055,-142.805,169.195,52.915,160.173
C05126=1013.811,284.806,-142.775,169.189,52.921,160.173
C05127=1013.806,284.558,-142.745,169.184,52.928,160.174
C05128=1013.800,284.310,-142.715,169.177,52.936,160.174
C05129=1013.794,284.062,-142.685,169.172,52.942,160.175
C05130=1013.789,283.814,-142.655,169.166,52.949,160.175
C05131=1013.783,283.566,-142.626,169.161,52.956,160.176
C05132=1013.778,283.318,-142.597,169.155,52.964,160.176
C05133=1013.772,283.069,-142.567,169.149,52.970,160.176
C05134=1013.766,282.822,-142.537,169.143,52.977,160.177
C05135=1013.760,282.573,-142.508,169.137,52.985,160.177
C05136=1013.755,282.325,-142.478,169.132,52.992,160.178
C05137=1013.750,282.077,-142.449,169.126,52.999,160.178
C05138=1013.743,281.829,-142.420,169.121,53.006,160.179
C05139=1013.738,281.581,-142.390,169.114,53.013,160.179
C05140=1013.732,281.332,-142.361,169.109,53.020,160.180
C05141=1013.727,281.084,-142.331,169.104,53.027,160.180
C05142=1013.721,280.836,-142.302,169.097,53.035,160.180
C05143=1013.716,280.588,-142.273,169.092,53.042,160.181
C05144=1013.710,280.339,-142.243,169.087,53.049,160.181
C05145=1013.704,280.091,-142.214,169.080,53.057,160.182
C05146=1013.698,279.843,-142.184,169.075,53.064,160.182
C05147=1013.694,279.595,-142.155,169.070,53.071,160.183
C05148=1013.688,279.347,-142.125,169.063,53.078,160.183
C05149=1013.682,279.099,-142.096,169.058,53.086,160.184
C05150=1013.677,278.851,-142.067,169.053,53.093,160.184
C05151=1013.671,278.602,-142.037,169.047,53.100,160.185
C05152=1013.666,278.351,-142.008,169.041,53.107,160.185
C05153=1013.660,278.100,-141.978,169.036,53.114,160.186
C05154=1013.654,277.849,-141.949,169.029,53.122,160.186
C05155=1013.649,277.598,-141.919,169.024,53.129,160.187
C05156=1013.643,277.349,-141.890,169.019,53.136,160.187
C05157=1013.638,277.102,-141.861,169.013,53.144,160.188
C05158=1013.632,276.853,-141.831,169.007,53.152,160.188
C05159=1013.627,276.604,-141.802,169.002,53.159,160.189
C05160=1013.622,276.356,-141.773,168.996,53.166,160.189
C05161=1013.616,276.108,-141.744,168.990,53.173,160.190
C05162=1013.611,275.861,-141.715,168.985,53.181,160.190
C05163=1013.605,275.612,-141.686,168.979,53.189,160.191
C05164=1013.599,275.363,-141.657,168.974,53.196,160.191
C05165=1013.594,275.116,-141.628,168.968,53.203,160.192
C05166=1013.589,274.867,-141.599,168.962,53.211,160.192
C05167=1013.583,274.619,-141.570,168.957,53.218,160.193
C05168=1013.578,274.370,-141.542,168.951,53.226,160.193
C05169=1013.572,274.123,-141.513,168.946,53.233,160.194
C05170=1013.567,273.874,-141.484,168.941,53.241,160.195
C05171=1013.561,273.626,-141.455,168.935,53.249,160.195
C05172=1013.555,273.378,-141.427,168.929,53.256,160.196
C05173=1013.550,273.129,-141.397,168.923,53.264,160.196
C05174=1013.544,272.881,-141.369,168.918,53.271,160.197
C05175=1013.539,272.633,-141.340,168.913,53.279,160.197
C05176=1013.534,272.385,-141.312,168.907,53.287,160.198
C05177=1013.528,272.136,-141.283,168.902,53.294,160.198
C05178=1013.523,271.888,-141.254,168.896,53.302,160.199
C05179=1013.518,271.639,-141.225,168.890,53.309,160.199
C05180=1013.512,271.392,-141.197,168.886,53.317,160.200
C05181=1013.506,271.143,-141.168,168.879,53.324,160.201
C05182=1013.501,270.895,-141.140,168.875,53.332,160.201
C05183=1013.496,270.647,-141.112,168.868,53.340,160.202
C05184=1013.490,270.398,-141.083,168.863,53.348,160.202
C05185=1013.485,270.150,-141.054,168.857,53.355,160.203
C05186=1013.479,269.901,-141.026,168.852,53.363,160.204
C05187=1013.474,269.653,-140.998,168.847,53.371,160.204
C05188=1013.468,269.405,-140.968,168.841,53.379,160.205
C05189=1013.463,269.157,-140.940,168.836,53.386,160.205
C05190=1013.458,268.908,-140.912,168.830,53.394,160.206
C05191=1013.452,268.660,-140.883,168.825,53.402,160.207
C05192=1013.447,268.412,-140.855,168.819,53.410,160.207
C05193=1013.442,268.164,-140.827,168.814,53.417,160.208
C05194=1013.436,267.915,-140.798,168.808,53.426,160.208
C05195=1013.431,267.667,-140.770,168.803,53.434,160.209
C05196=1013.426,267.419,-140.742,168.797,53.442,160.210
C05197=1013.420,267.170,-140.714,168.792,53.449,160.210
C05198=1013.414,266.922,-140.686,168.786,53.457,160.211
C05199=1013.409,266.674,-140.658,168.782,53.465,160.212
C05200=1013.404,266.425,-140.629,168.776,53.473,160.212
C05201=1013.398,266.177,-140.601,168.771,53.481,160.213
C05202=1013.393,265.929,-140.573,168.765,53.489,160.213
C05203=1013.387,265.680,-140.545,168.760,53.497,160.214
C05204=1013.382,265.432,-140.517,168.754,53.505,160.215
C05205=1013.378,265.183,-140.489,168.749,53.513,160.215
C05206=1013.372,264.935,-140.461,168.743,53.521,160.216
C05207=1013.366,264.686,-140.432,168.739,53.529,160.217
C05208=1013.361,264.439,-140.405,168.733,53.537,160.217
C05209=1013.355,264.192,-140.377,168.728,53.545,160.218
C05210=1013.350,263.945,-140.349,168.722,53.553,160.218
C05211=1013.345,263.697,-140.321,168.717,53.561,160.219
C05212=1013.339,263.450,-140.294,168.711,53.569,160.220
C05213=1013.334,263.202,-140.266,168.706,53.577,160.221
C05214=1013.329,262.955,-140.238,168.700,53.585,160.221
C05215=1013.324,262.708,-140.211,168.696,53.593,160.222
C05216=1013.318,262.459,-140.183,168.690,53.601,160.222
C05217=1013.312,262.211,-140.155,168.685,53.609,160.223
C05218=1013.307,261.962,-140.127,168.679,53.618,160.224
C05219=1013.302,261.714,-140.100,168.675,53.626,160.225
C05220=1013.297,261.466,-140.072,168.669,53.635,160.225
C05221=1013.292,261.218,-140.044,168.664,53.642,160.226
C05222=1013.286,260.969,-140.016,168.658,53.651,160.227
C05223=1013.281,260.720,-139.989,168.653,53.659,160.227
C05224=1013.275,260.472,-139.961,168.648,53.667,160.228
C05225=1013.271,260.223,-139.933,168.642,53.675,160.229
C05226=1013.266,259.975,-139.905,168.637,53.683,160.229
C05227=1013.260,259.727,-139.877,168.632,53.692,160.230
C05228=1013.255,259.478,-139.850,168.627,53.700,160.231
C05229=1013.249,259.231,-139.822,168.621,53.708,160.232
C05230=1013.244,258.982,-139.795,168.615,53.717,160.232
C05231=1013.239,258.733,-139.768,168.611,53.725,160.233
C05232=1013.233,258.486,-139.741,168.605,53.734,160.234
C05233=1013.228,258.237,-139.713,168.600,53.742,160.235
C05234=1013.222,257.988,-139.686,168.594,53.751,160.235
C05235=1013.217,257.739,-139.659,168.590,53.759,160.236
C05236=1013.212,257.490,-139.632,168.584,53.768,160.237
C05237=1013.205,257.243,-139.604,168.578,53.776,160.238
C05238=1013.200,256.994,-139.577,168.574,53.784,160.238
C05239=1013.195,256.746,-139.551,168.568,53.793,160.239
C05240=1013.190,256.497,-139.523,168.563,53.802,160.240
C05241=1013.185,256.248,-139.496,168.558,53.810,160.241
C05242=1013.179,256.000,-139.469,168.552,53.819,160.241
C05243=1013.173,255.752,-139.441,168.547,53.828,160.242
C05244=1013.168,255.504,-139.415,168.541,53.836,160.243
C05245=1013.163,255.255,-139.388,168.537,53.845,160.244
C05246=1013.158,255.006,-139.360,168.531,53.853,160.244
C05247=1013.152,254.758,-139.334,168.526,53.862,160.245
C05248=1013.147,254.509,-139.306,168.521,53.870,160.246
C05249=1013.141,254.261,-139.280,168.516,53.879,160.247
C05250=1013.136,254.012,-139.253,168.510,53.887,160.247
C05251=1013.130,253.764,-139.226,168.505,53.896,160.248
C05252=1013.125,253.515,-139.199,168.501,53.905,160.249
C05253=1013.121,253.267,-139.172,168.495,53.913,160.250
C05254=1013.115,253.019,-139.145,168.490,53.922,160.251
C05255=1013.110,252.770,-139.118,168.484,53.931,160.251
C05256=1013.104,252.522,-139.091,168.480,53.939,160.252
C05257=1013.099,252.273,-139.064,168.474,53.948,160.253
C05258=1013.094,252.024,-139.037,168.468,53.957,160.254
C05259=1013.088,251.776,-139.010,168.464,53.965,160.255
C05260=1013.083,251.527,-138.983,168.459,53.974,160.256
C05261=1013.078,251.278,-138.957,168.453,53.983,160.256
C05262=1013.073,251.031,-138.930,168.448,53.992,160.257
C05263=1013.068,250.782,-138.903,168.443,54.001,160.258
C05264=1013.063,250.533,-138.876,168.438,54.010,160.259
C05265=1013.058,250.285,-138.849,168.433,54.018,160.259
C05266=1013.052,250.036,-138.822,168.427,54.027,160.260
C05267=1013.048,249.788,-138.796,168.422,54.036,160.261
C05268=1013.042,249.540,-138.769,168.418,54.045,160.262
C05269=1013.037,249.291,-138.742,168.412,54.053,160.263
C05270=1013.032,249.043,-138.716,168.407,54.062,160.264
C05271=1013.027,248.795,-138.689,168.402,54.071,160.264
C05272=1013.022,248.546,-138.661,168.397,54.080,160.265
C05273=1013.016,248.298,-138.635,168.392,54.089,160.266
C05274=1013.012,248.049,-138.609,168.386,54.097,160.267
C05275=1013.004,247.710,-138.572,168.379,54.110,160.268
C05276=1013.131,265.964,-140.941,168.732,53.611,160.234
C05277=1013.136,266.178,-140.965,168.736,53.605,160.233
C05278=1013.141,266.393,-140.990,168.741,53.597,160.233
C05279=1013.145,266.607,-141.014,168.746,53.590,160.232
C05280=1013.149,266.822,-141.039,168.750,53.584,160.231
C05281=1013.154,267.036,-141.062,168.755,53.576,160.231
C05282=1013.159,267.250,-141.087,168.760,53.570,160.231
C05283=1013.164,267.465,-141.111,168.764,53.563,160.230
C05284=1013.168,267.679,-141.135,168.769,53.556,160.229
C05285=1013.174,267.927,-141.163,168.774,53.548,160.229
C05286=1013.179,268.175,-141.192,168.780,53.540,160.228
C05287=1013.185,268.423,-141.221,168.785,53.533,160.228
C05288=1013.190,268.672,-141.249,168.791,53.525,160.227
C05289=1013.195,268.920,-141.277,168.796,53.517,160.226
C05290=1013.201,269.169,-141.305,168.802,53.509,160.226
C05291=1013.206,269.417,-141.333,168.807,53.501,160.225
C05292=1013.211,269.665,-141.361,168.813,53.493,160.224
C05293=1013.216,269.914,-141.390,168.818,53.486,160.224
C05294=1013.222,270.161,-141.419,168.824,53.477,160.223
C05295=1013.227,270.410,-141.447,168.829,53.470,160.223
C05296=1013.233,270.658,-141.476,168.835,53.462,160.222
C05297=1013.238,270.906,-141.504,168.840,53.454,160.221
C05298=1013.243,271.155,-141.533,168.846,53.447,160.221
C05299=1013.249,271.403,-141.561,168.851,53.439,160.220
C05300=1013.255,271.652,-141.590,168.857,53.431,160.220
C05301=1013.259,271.900,-141.618,168.862,53.423,160.219
C05302=1013.265,272.147,-141.647,168.868,53.416,160.219
C05303=1013.270,272.396,-141.676,168.873,53.408,160.218
C05304=1013.276,272.645,-141.704,168.880,53.400,160.218
C05305=1013.281,272.893,-141.733,168.884,53.392,160.217
C05306=1013.286,273.141,-141.761,168.891,53.385,160.217
C05307=1013.292,273.389,-141.791,168.896,53.378,160.216
C05308=1013.297,273.638,-141.819,168.901,53.370,160.215
C05309=1013.303,273.886,-141.847,168.907,53.362,160.215
C05310=1013.308,274.134,-141.877,168.912,53.354,160.214
C05311=1013.314,274.383,-141.905,168.918,53.347,160.214
C05312=1013.319,274.631,-141.934,168.924,53.340,160.213
C05313=1013.325,274.879,-141.963,168.929,53.331,160.213
C05314=1013.330,275.127,-141.992,168.935,53.324,160.212
C05315=1013.336,275.376,-142.020,168.941,53.317,160.212
C05316=1013.341,275.624,-142.050,168.946,53.309,160.211
C05317=1013.347,275.872,-142.078,168.951,53.302,160.210
C05318=1013.352,276.121,-142.107,168.957,53.294,160.210
C05319=1013.358,276.368,-142.136,168.963,53.287,160.210
C05320=1013.363,276.617,-142.166,168.969,53.279,160.209
C05321=1013.368,276.865,-142.194,168.974,53.271,160.208
C05322=1013.373,277.113,-142.224,168.979,53.264,160.208
C05323=1013.380,277.361,-142.253,168.986,53.257,160.208
C05324=1013.385,277.609,-142.282,168.991,53.250,160.207
C05325=1013.390,277.863,-142.312,168.997,53.242,160.207
C05326=1013.396,278.116,-142.341,169.002,53.234,160.206
C05327=1013.401,278.370,-142.372,169.008,53.227,160.205
C05328=1013.407,278.623,-142.401,169.014,53.219,160.205
C05329=1013.412,278.871,-142.430,169.020,53.212,160.205
C05330=1013.418,279.119,-142.460,169.025,53.205,160.204
C05331=1013.423,279.368,-142.490,169.032,53.197,160.204
C05332=1013.429,279.616,-142.518,169.037,53.190,160.203
C05333=1013.434,279.864,-142.547,169.042,53.183,160.203
C05334=1013.440,280.113,-142.577,169.049,53.175,160.202
C05335=1013.446,280.361,-142.606,169.054,53.168,160.202
C05336=1013.451,280.609,-142.635,169.059,53.161,160.201
C05337=1013.456,280.857,-142.665,169.065,53.154,160.201
C05338=1013.462,281.105,-142.695,169.071,53.146,160.200
C05339=1013.468,281.354,-142.724,169.077,53.139,160.200
C05340=1013.473,281.601,-142.753,169.082,53.132,160.199
C05341=1013.479,281.850,-142.782,169.088,53.125,160.199
C05342=1013.485,282.098,-142.811,169.094,53.117,160.198
C05343=1013.490,282.346,-142.841,169.099,53.110,160.198
C05344=1013.496,282.595,-142.871,169.105,53.104,160.198
C05345=1013.501,282.842,-142.900,169.112,53.096,160.197
C05346=1013.507,283.090,-142.930,169.117,53.089,160.197
C05347=1013.513,283.338,-142.959,169.122,53.082,160.196
